(* IEC 61131-3 sources: F100R_S278_Temperville/MyController.device.xml.v3^/Plc Logic.plclogic.xml.v3^/Application.application.xml.v3^/02_Operação (part 3) *)

(* ---- K_Guilhotina01Inf.prg.st ---- *)
PROGRAM K_Guilhotina01Inf
VAR
	PassoHomeGuilhotina01Inf: INT;
	PassoAjusteGuilhotina01Inf: INT;
	PassoPausaHomeGuilhotina01Inf: INT;
	PassoPausaAjusteGuilhotina01Inf: INT;
	PassoAlmHomeGuilhotina01Inf: INT;
	PassoAlmAjusteGuilhotina01Inf: INT;
	///Bloco Converte Milimetro em Pulsos
	ConversorMilimPul01Guilho01Inf: MmConversorPulso;
	///Bloco Converte Milimetro em Pulsos
	ConversorMilimPul02Guilho01Inf: MmConversorPulso;
	///Bloco Converte Pulsos em Milimetros
	ConversorPulMilimGuilho01Inf: PulsoConversorMm;
	xSetValorSpAltGuil01InfSup: BOOL;
	iAlturaGhilhotina01InfAux: INT;
	xAjustarAlturaGuilhotina01Inf: BOOL;
	iVelocidadeHomeGuilhotina01Inf: INT;
	iVelocidadeGuilhotina01Inf: INT;
	dValEncoAlturaGuilhotina01Inf: DINT;
	dValEncoToleranciaGuilhotina01Inf: DINT;
	dValEncoAlturaVelMinGuilhotina01Inf: DINT;
	xAbreJogGuilhotina01Inf: BOOL;
	xFechaJogGuilhotina01Inf: BOOL;
	xAbreGuilhotina01Inf: BOOL;
	xFechaGuilhotina01Inf: BOOL;
END_VAR

IF iAlturaGhilhotina01Inf <> iAlturaGhilhotina01InfAux THEN
	xSetValorSpAltGuil01InfSup:=TRUE;

END_IF;

IF xSetValorSpAltGuil01InfSup THEN
	iAlturaGhilhotina01InfAux:=iAlturaGhilhotina01Inf;
ELSE
	IF NOT xMotorGuilhotina01InfLigado THEN
		iAlturaGhilhotina01Inf:=iAlturaAtualGuilhotina01Inf;
	END_IF;
END_IF

IF iAlturaGhilhotina01InfAux=iAlturaAtualGuilhotina01Inf THEN
	xSetValorSpAltGuil01InfSup:=FALSE;
END_IF

// CONVERSÃO MILIMETROS EM PULSOS

ConversorMilimPul01Guilho01Inf(
	dPulso:= 105563,
	dMilimetro:= 100,
	iEntrMilimetro01:= iAlturaGhilhotina01InfAux,//iAlturaGhilhotina02,
	dSaidaPulso01=> dValEncoAlturaGuilhotina01Inf);

ConversorMilimPul02Guilho01Inf(
	dPulso:= 105563,
	dMilimetro:= 100,
	iEntrMilimetro01:= 2,//iValEncoToleranciaGuilhotina,
	iEntrMilimetro02:= 8,//iValEncoAlturaVelMinGuilhotina,
	dSaidaPulso01=> dValEncoToleranciaGuilhotina01Inf,
	dSaidaPulso02=> dValEncoAlturaVelMinGuilhotina01Inf);

// SEQUENCIA DE HOME

CASE PassoHomeGuilhotina01Inf OF

		0:	IF xIniciaHomeGuilhotina01Inf THEN
				PassoHomeGuilhotina01Inf:=10;
			END_IF

		10:	xIniciaHomeGuilhotina01Inf:=FALSE;
			xHomeGuilhotina01InfOk:=FALSE;
			xAjusteAlturaGuilhotina01InfOK:=FALSE;
			xGuilhotina01InfEmHome:=TRUE;
			iVelocidadeGuilhotina01Inf:= 300;//1*iVelocidadeHomeDuctosResfrSup02;
			PassoHomeGuilhotina01Inf:=15;

		15: xFechaGuilhotina01Inf:=TRUE;
			PassoHomeGuilhotina01Inf:=20;

		20:	IF xSensorFechadoGuilhotina01Inf THEN
				PassoHomeGuilhotina01Inf:=50;
			END_IF
			IF xPause THEN
				PassoPausaHomeGuilhotina01Inf:=10;
				PassoHomeGuilhotina01Inf:=300;
			END_IF
			IF xAlarmeMotorGuilhotina01Inf THEN
				PassoAlmHomeGuilhotina01Inf:=10;
				PassoHomeGuilhotina01Inf:=400;
			END_IF

		50:	xFechaGuilhotina01Inf:=FALSE;
			PassoHomeGuilhotina01Inf:=55;

		55:	iVelocidadeGuilhotina01Inf:= 50;
			PassoHomeGuilhotina01Inf:=56;

		56:	xAbreGuilhotina01Inf:=TRUE;
			PassoHomeGuilhotina01Inf:=60;

		60:	IF NOT xSensorFechadoGuilhotina01Inf THEN
				PassoHomeGuilhotina01Inf:=70;
			END_IF
			IF xPause THEN
				PassoPausaHomeGuilhotina01Inf:=50;
				PassoHomeGuilhotina01Inf:=300;
			END_IF
			IF xAlarmeMotorGuilhotina01Inf THEN
				PassoAlmHomeGuilhotina01Inf:=50;
				PassoHomeGuilhotina01Inf:=400;
			END_IF

		70:	xAbreGuilhotina01Inf:=FALSE;
			PassoHomeGuilhotina01Inf:=74;

		74:	IF NOT xMotorGuilhotina01InfLigado THEN
				PassoHomeGuilhotina01Inf:=75;
			END_IF

		75: xHomeEncoderGuilhotinaResfriador01Inf:=TRUE;
			PassoHomeGuilhotina01Inf:=80;

		80: xHomeEncoderGuilhotinaResfriador01Inf:=FALSE;
			xGuilhotina01InfEmHome:=FALSE;
			xHomeGuilhotina01InfOk:=TRUE;

		// Emergência Pausa/Reinicio
		300:xAbreGuilhotina01Inf:=FALSE;
			xAbreGuilhotina01Inf:=FALSE;
			PassoHomeGuilhotina01Inf:=301;

		301:xDuctosSup02EmHome:=FALSE;
			PassoHomeGuilhotina01Inf:=302;

		302:IF xRestart THEN
				PassoHomeGuilhotina01Inf:=303;
			END_IF

		303:PassoHomeGuilhotina01Inf:=0;//PassoPausaHomeDuctosResfrSup02;

		// Alarme Motor Parada/Reinicio
		400:xFechaGuilhotina01Inf:=FALSE;
			xAbreGuilhotina01Inf:=FALSE;
			PassoHomeGuilhotina01Inf:=401;

		401:PassoHomeGuilhotina01Inf:=402;

		402:IF xRestart AND iCanOpenInverGuilResfr01InfStateOk THEN
				PassoHomeGuilhotina01Inf:=PassoAlmHomeGuilhotina01Inf;
			END_IF
END_CASE

// SEQUENCIA DE FUNCIONAMENTO

IF (xBtRecAjustaGuilhotina01Inf OR BtParamGuilhotina01Inf) AND xHomeGuilhotina01InfOk THEN
	xAjustarAlturaGuilhotina01Inf:=TRUE;
	xBtRecAjustaGuilhotina01Inf:=FALSE;
	BtParamGuilhotina01Inf:=FALSE;
ELSE
	xBtRecAjustaGuilhotina01Inf:=FALSE;
	BtParamGuilhotina01Inf:=FALSE;
END_IF

CASE PassoAjusteGuilhotina01Inf OF

		0:	IF xAjustarAlturaGuilhotina01Inf THEN
				PassoAjusteGuilhotina01Inf:=10;
			END_IF

		10:	xAjustarAlturaGuilhotina01Inf:=FALSE;
			xAjusteAlturaGuilhotina01InfOK:=FALSE;
			xGuilhotina01InfEmAjuste:=TRUE;
			IF (dValorEncoderGuilhotinaResfriador01Inf>=dValEncoAlturaGuilhotina01Inf-dValEncoToleranciaGuilhotina01Inf) AND (dValorEncoderGuilhotinaResfriador01Inf<=dValEncoAlturaGuilhotina01Inf+dValEncoToleranciaGuilhotina01Inf) THEN
				PassoAjusteGuilhotina01Inf:=180;//Não se Move
			END_IF
			IF dValorEncoderGuilhotinaResfriador01Inf<dValEncoAlturaGuilhotina01Inf-dValEncoToleranciaGuilhotina01Inf THEN
				PassoAjusteGuilhotina01Inf:=20;//Sobe
			END_IF
			IF dValorEncoderGuilhotinaResfriador01Inf>dValEncoAlturaGuilhotina01Inf+dValEncoToleranciaGuilhotina01Inf THEN
				PassoAjusteGuilhotina01Inf:=100;//Desce
			END_IF

//Sobe

		20:	iVelocidadeGuilhotina01Inf:= iVelocidadeAjusteGuilhotina01Inf;
			PassoAjusteGuilhotina01Inf:=25;

		25: xAbreGuilhotina01Inf:=TRUE;
			PassoAjusteGuilhotina01Inf:=30;

		30:	IF dValorEncoderGuilhotinaResfriador01Inf>=dValEncoAlturaGuilhotina01Inf-dValEncoAlturaVelMinGuilhotina01Inf THEN
				PassoAjusteGuilhotina01Inf:=40;
			END_IF
			IF iVelocidadeGuilhotina01Inf<> iVelocidadeAjusteGuilhotina01Inf THEN
				PassoAjusteGuilhotina01Inf:=20;
			END_IF
			IF xSensorAbertoGuilhotina01Inf THEN
				PassoAjusteGuilhotina01Inf:=200;
			END_IF

			IF xPause THEN
				PassoPausaAjusteGuilhotina01Inf:=20;
				PassoAjusteGuilhotina01Inf:=300;
			END_IF
			IF xAlarmeMotorGuilhotina01Inf THEN
				PassoAlmAjusteGuilhotina01Inf:=20;
				PassoAjusteGuilhotina01Inf:=400;
			END_IF

		40:	iVelocidadeGuilhotina01Inf:= iVelocidadeMinimaGuilhotina01Inf;
			PassoAjusteGuilhotina01Inf:=50;

		50:	IF dValorEncoderGuilhotinaResfriador01Inf>=dValEncoAlturaGuilhotina01Inf THEN
				PassoAjusteGuilhotina01Inf:=60;
			END_IF
			IF iVelocidadeGuilhotina01Inf<> iVelocidadeMinimaGuilhotina01Inf THEN
				PassoAjusteGuilhotina01Inf:=40;
			END_IF
			IF xPause THEN
				PassoPausaAjusteGuilhotina01Inf:=40;
				PassoAjusteGuilhotina01Inf:=300;
			END_IF
			IF xAlarmeMotorGuilhotina01Inf THEN
				PassoAlmAjusteGuilhotina01Inf:=40;
				PassoAjusteGuilhotina01Inf:=400;
			END_IF

		60: xAbreGuilhotina01Inf:=FALSE;
			PassoAjusteGuilhotina01Inf:=180;
//Desce

		100:iVelocidadeGuilhotina01Inf:= 1*iVelocidadeAjusteGuilhotina01Inf;
			PassoAjusteGuilhotina01Inf:=105;

		105:xFechaGuilhotina01Inf:=TRUE;
			PassoAjusteGuilhotina01Inf:=110;

		110:IF dValorEncoderGuilhotinaResfriador01Inf<dValEncoAlturaGuilhotina01Inf+dValEncoAlturaVelMinGuilhotina01Inf THEN
				PassoAjusteGuilhotina01Inf:=120;
			END_IF
			IF iVelocidadeGuilhotina01Inf<> 1*iVelocidadeAjusteGuilhotina01Inf THEN
				PassoAjusteGuilhotina01Inf:=100;
			END_IF
			IF	xSensorFechadoGuilhotina01Inf THEN
				PassoAjusteGuilhotina01Inf:=200;
			END_IF
			IF xPause THEN
				PassoPausaAjusteGuilhotina01Inf:=100;
				PassoAjusteGuilhotina01Inf:=300;
			END_IF
			IF xAlarmeMotorGuilhotina01Inf THEN
				PassoAlmAjusteGuilhotina01Inf:=100;
				PassoAjusteGuilhotina01Inf:=400;
			END_IF

		120:iVelocidadeGuilhotina01Inf:= 1*iVelocidadeMinimaGuilhotina01Inf;
			PassoAjusteGuilhotina01Inf:=130;

		130:IF  dValorEncoderGuilhotinaResfriador01Inf<=dValEncoAlturaGuilhotina01Inf THEN
				PassoAjusteGuilhotina01Inf:=140;
			END_IF
			IF xPause THEN
				PassoPausaAjusteGuilhotina01Inf:=120;
				PassoAjusteGuilhotina01Inf:=300;
			END_IF
			IF xAlarmeMotorGuilhotina01Inf THEN
				PassoAlmAjusteGuilhotina01Inf:=120;
				PassoAjusteGuilhotina01Inf:=400;
			END_IF

		140:xFechaGuilhotina01Inf:=FALSE;
			PassoAjusteGuilhotina01Inf:=180;
//Fim

		180:xAjusteAlturaGuilhotina01InfOK:=TRUE;
			xGuilhotina01InfEmAjuste:=FALSE;
			PassoAjusteGuilhotina01Inf:=0;

		200:xAbreGuilhotina01Inf:=FALSE;
			xFechaGuilhotina01Inf:=FALSE;
			PassoAjusteGuilhotina01Inf:=0;

		// Emergência Pausa/Reinicio
		300:xAbreGuilhotina01Inf:=FALSE;
			xFechaGuilhotina01Inf:=FALSE;
			PassoAjusteGuilhotina01Inf:=301;

		301:PassoAjusteGuilhotina01Inf:=302;

		302:IF xRestart THEN
				PassoAjusteGuilhotina01Inf:=303;
			END_IF

		303: PassoAjusteGuilhotina01Inf:=PassoPausaAjusteGuilhotina01Inf;

		// Alarme Motor Parada/Reinicio
		400:xAbreGuilhotina01Inf:=FALSE;
			xFechaGuilhotina01Inf:=FALSE;
			PassoAjusteGuilhotina01Inf:=401;

		401:PassoAjusteGuilhotina01Inf:=402;

		402:IF xRestart AND iCanOpenInverGuilResfr01InfStateOk THEN
				PassoAjusteGuilhotina01Inf:=PassoAlmAjusteGuilhotina01Inf;
			END_IF

END_CASE

// MOVIMENTAÇÃO PELO COMANDO ENTRADAS DIGITAIS DO INVERSOR
// Comando e Dirreção
xMotorGuilhotina01InfAbre:= xAbreGuilhotina01Inf OR xAbreJogGuilhotina01Inf;
xMotorGuilhotina01InfFecha:= xFechaGuilhotina01Inf OR xFechaJogGuilhotina01Inf;

InversorGuilhot01Inf.i_xAvanco:=xMotorGuilhotina01InfAbre;
InversorGuilhot01Inf.i_xRecuo:=xMotorGuilhotina01InfFecha;

// Velocidade
InversorGuilhot01Inf.i_iFreqRef:=iVelocidadeGuilhotina01Inf;
//---------------------------------------------------------------------------------\\

ConversorPulMilimGuilho01Inf(
	dPulso:=105563,
	dMilimetro:= 100,
	dEntradaPulso01:= dValorEncoderGuilhotinaResfriador01Inf,
	iSaidaMilimetro01=> iAlturaAtualGuilhotina01Inf );

IF xOperacaoManual THEN
	PassoHomeGuilhotina01Inf:=0;
	PassoAjusteGuilhotina01Inf:=0;
	xIniciaHomeGuilhotina01Inf:=FALSE;
	xAjusteAlturaGuilhotina01InfOK:=FALSE;
	xGuilhotina01InfEmHome:=FALSE;
	xGuilhotina01InfEmAjuste:=FALSE;

	xAbreGuilhotina01Inf:=FALSE;
	xFechaGuilhotina01Inf:=FALSE;
END_IF

(*-------------------- Manual Jog--------------------------*)

(* ---- K_Guilhotina01Sup.prg.st ---- *)
PROGRAM K_Guilhotina01Sup
VAR
	PassoHomeGuilhotina01Sup: INT;
	PassoAjusteGuilhotina01Sup: INT;
	PassoPausaHomeGuilhotina01Sup: INT;
	PassoPausaAjusteGuilhotina01Sup: INT;
	PassoAlmHomeGuilhotina01Sup: INT;
	PassoAlmAjusteGuilhotina01Sup: INT;
	///Bloco Converte Milimetro em Pulsos
	ConversorMilimPul01Guilho01Sup: MmConversorPulso;
	///Bloco Converte Milimetro em Pulsos
	ConversorMilimPul02Guilho01Sup: MmConversorPulso;
	///Bloco Converte Pulsos em Milimetros
	ConversorPulMilimGuilho01Sup: PulsoConversorMm;
	xSetValorSpAltGuil01SupSup: BOOL;
	iAlturaGhilhotina01SupAux: INT;
	xAjustarAlturaGuilhotina01Sup: BOOL;
	iVelocidadeHomeGuilhotina01Sup: INT;
	iVelocidadeGuilhotina01Sup: INT;
	dValEncoAlturaGuilhotina01Sup: DINT;
	dValEncoToleranciaGuilhotina01Sup: DINT;
	dValEncoAlturaVelMinGuilhotina01Sup: DINT;
	xAbreJogGuilhotina01Sup: BOOL;
	xFechaJogGuilhotina01Sup: BOOL;
	xAbreGuilhotina01Sup: BOOL;
	xFechaGuilhotina01Sup: BOOL;
END_VAR

IF iAlturaGhilhotina01Sup <> iAlturaGhilhotina01SupAux THEN
	xSetValorSpAltGuil01SupSup:=TRUE;

END_IF;

IF xSetValorSpAltGuil01SupSup THEN
	iAlturaGhilhotina01SupAux:=iAlturaGhilhotina01Sup;
ELSE
	IF NOT xMotorGuilhotina01SupLigado THEN
		iAlturaGhilhotina01Sup:=iAlturaAtualGuilhotina01Sup;
	END_IF;
END_IF

IF iAlturaGhilhotina01SupAux=iAlturaAtualGuilhotina01Sup THEN
	xSetValorSpAltGuil01SupSup:=FALSE;
END_IF

// CONVERSÃO MILIMETROS EM PULSOS

ConversorMilimPul01Guilho01Sup(
	dPulso:= 107918,
	dMilimetro:= 100,
	iEntrMilimetro01:= iAlturaGhilhotina01SupAux,//iAlturaGhilhotina02,
	dSaidaPulso01=> dValEncoAlturaGuilhotina01Sup);

ConversorMilimPul02Guilho01Sup(
	dPulso:= 107918,
	dMilimetro:= 100,
	iEntrMilimetro01:= 2,//iValEncoToleranciaGuilhotina,
	iEntrMilimetro02:= 8,//iValEncoAlturaVelMinGuilhotina,
	dSaidaPulso01=> dValEncoToleranciaGuilhotina01Sup,
	dSaidaPulso02=> dValEncoAlturaVelMinGuilhotina01Sup);

// SEQUENCIA DE HOME

CASE PassoHomeGuilhotina01Sup OF

		0:	IF xIniciaHomeGuilhotina01Sup THEN
				PassoHomeGuilhotina01Sup:=10;
			END_IF

		10:	xIniciaHomeGuilhotina01Sup:=FALSE;
			xHomeGuilhotina01SupOk:=FALSE;
			xAjusteAlturaGuilhotina01SupOK:=FALSE;
			xGuilhotina01SupEmHome:=TRUE;
			iVelocidadeGuilhotina01Sup:= 300;//1*iVelocidadeHomeDuctosResfrSup02;
			PassoHomeGuilhotina01Sup:=15;

		15: xFechaGuilhotina01Sup:=TRUE;
			PassoHomeGuilhotina01Sup:=20;

		20:	IF xSensorFechadoGuilhotina01Sup THEN
				PassoHomeGuilhotina01Sup:=50;
			END_IF
			IF xPause THEN
				PassoPausaHomeGuilhotina01Sup:=10;
				PassoHomeGuilhotina01Sup:=300;
			END_IF
			IF xAlarmeMotorGuilhotina01Sup THEN
				PassoAlmHomeGuilhotina01Sup:=10;
				PassoHomeGuilhotina01Sup:=400;
			END_IF

		50:	xFechaGuilhotina01Sup:=FALSE;
			PassoHomeGuilhotina01Sup:=55;

		55:	iVelocidadeGuilhotina01Sup:= 50;
			PassoHomeGuilhotina01Sup:=56;

		56:	xAbreGuilhotina01Sup:=TRUE;
			PassoHomeGuilhotina01Sup:=60;

		60:	IF NOT xSensorFechadoGuilhotina01Sup THEN
				PassoHomeGuilhotina01Sup:=70;
			END_IF
			IF xPause THEN
				PassoPausaHomeGuilhotina01Sup:=50;
				PassoHomeGuilhotina01Sup:=300;
			END_IF
			IF xAlarmeMotorGuilhotina01Sup THEN
				PassoAlmHomeGuilhotina01Sup:=50;
				PassoHomeGuilhotina01Sup:=400;
			END_IF

		70:	xAbreGuilhotina01Sup:=FALSE;
			PassoHomeGuilhotina01Sup:=74;

		74:	IF NOT xMotorGuilhotina01SupLigado THEN
				PassoHomeGuilhotina01Sup:=75;
			END_IF

		75: xHomeEncoderGuilhotinaResfriador01Sup:=TRUE;
			PassoHomeGuilhotina01Sup:=80;

		80: xHomeEncoderGuilhotinaResfriador01Sup:=FALSE;
			xGuilhotina01SupEmHome:=FALSE;
			xHomeGuilhotina01SupOk:=TRUE;

		// Emergência Pausa/Reinicio
		300:xAbreGuilhotina01Sup:=FALSE;
			xAbreGuilhotina01Sup:=FALSE;
			PassoHomeGuilhotina01Sup:=301;

		301:xDuctosSup02EmHome:=FALSE;
			PassoHomeGuilhotina01Sup:=302;

		302:IF xRestart THEN
				PassoHomeGuilhotina01Sup:=303;
			END_IF

		303:PassoHomeGuilhotina01Sup:=0;//PassoPausaHomeDuctosResfrSup02;

		// Alarme Motor Parada/Reinicio
		400:xFechaGuilhotina01Sup:=FALSE;
			xAbreGuilhotina01Sup:=FALSE;
			PassoHomeGuilhotina01Sup:=401;

		401:PassoHomeGuilhotina01Sup:=402;

		402:IF xRestart AND iCanOpenInverGuilResfr01SupStateOk THEN
				PassoHomeGuilhotina01Sup:=PassoAlmHomeGuilhotina01Sup;
			END_IF
END_CASE

// SEQUENCIA DE FUNCIONAMENTO

IF (xBtRecAjustaGuilhotina01Sup OR BtParamGuilhotina01Sup) AND xHomeGuilhotina01SupOk THEN
	xAjustarAlturaGuilhotina01Sup:=TRUE;
	xBtRecAjustaGuilhotina01Sup:=FALSE;
	BtParamGuilhotina01Sup:=FALSE;
ELSE
	xBtRecAjustaGuilhotina01Sup:=FALSE;
	BtParamGuilhotina01Sup:=FALSE;
END_IF

CASE PassoAjusteGuilhotina01Sup OF

		0:	IF xAjustarAlturaGuilhotina01Sup THEN
				PassoAjusteGuilhotina01Sup:=10;
			END_IF

		10:	xAjustarAlturaGuilhotina01Sup:=FALSE;
			xAjusteAlturaGuilhotina01SupOK:=FALSE;
			xGuilhotina01SupEmAjuste:=TRUE;
			IF (dValorEncoderGuilhotinaResfriador01Sup>=dValEncoAlturaGuilhotina01Sup-dValEncoToleranciaGuilhotina01Sup) AND (dValorEncoderGuilhotinaResfriador01Sup<=dValEncoAlturaGuilhotina01Sup+dValEncoToleranciaGuilhotina01Sup) THEN
				PassoAjusteGuilhotina01Sup:=180;//Não se Move
			END_IF
			IF dValorEncoderGuilhotinaResfriador01Sup<dValEncoAlturaGuilhotina01Sup-dValEncoToleranciaGuilhotina01Sup THEN
				PassoAjusteGuilhotina01Sup:=20;//Sobe
			END_IF
			IF dValorEncoderGuilhotinaResfriador01Sup>dValEncoAlturaGuilhotina01Sup+dValEncoToleranciaGuilhotina01Sup THEN
				PassoAjusteGuilhotina01Sup:=100;//Desce
			END_IF

//Sobe

		20:	iVelocidadeGuilhotina01Sup:= iVelocidadeAjusteGuilhotina01Sup;
			PassoAjusteGuilhotina01Sup:=25;

		25: xAbreGuilhotina01Sup:=TRUE;
			PassoAjusteGuilhotina01Sup:=30;

		30:	IF dValorEncoderGuilhotinaResfriador01Sup>=dValEncoAlturaGuilhotina01Sup-dValEncoAlturaVelMinGuilhotina01Sup THEN
				PassoAjusteGuilhotina01Sup:=40;
			END_IF
			IF iVelocidadeGuilhotina01Sup<> iVelocidadeAjusteGuilhotina01Sup THEN
				PassoAjusteGuilhotina01Sup:=20;
			END_IF
			IF xSensorAbertoGuilhotina01Sup THEN
				PassoAjusteGuilhotina01Sup:=200;
			END_IF

			IF xPause THEN
				PassoPausaAjusteGuilhotina01Sup:=20;
				PassoAjusteGuilhotina01Sup:=300;
			END_IF
			IF xAlarmeMotorGuilhotina01Sup THEN
				PassoAlmAjusteGuilhotina01Sup:=20;
				PassoAjusteGuilhotina01Sup:=400;
			END_IF

		40:	iVelocidadeGuilhotina01Sup:= iVelocidadeMinimaGuilhotina01Sup;
			PassoAjusteGuilhotina01Sup:=50;

		50:	IF dValorEncoderGuilhotinaResfriador01Sup>=dValEncoAlturaGuilhotina01Sup THEN
				PassoAjusteGuilhotina01Sup:=60;
			END_IF
			IF iVelocidadeGuilhotina01Sup<> iVelocidadeMinimaGuilhotina01Sup THEN
				PassoAjusteGuilhotina01Sup:=40;
			END_IF
			IF xPause THEN
				PassoPausaAjusteGuilhotina01Sup:=40;
				PassoAjusteGuilhotina01Sup:=300;
			END_IF
			IF xAlarmeMotorGuilhotina01Sup THEN
				PassoAlmAjusteGuilhotina01Sup:=40;
				PassoAjusteGuilhotina01Sup:=400;
			END_IF

		60: xAbreGuilhotina01Sup:=FALSE;
			PassoAjusteGuilhotina01Sup:=180;
//Desce

		100:iVelocidadeGuilhotina01Sup:= 1*iVelocidadeAjusteGuilhotina01Sup;
			PassoAjusteGuilhotina01Sup:=105;

		105:xFechaGuilhotina01Sup:=TRUE;
			PassoAjusteGuilhotina01Sup:=110;

		110:IF dValorEncoderGuilhotinaResfriador01Sup<dValEncoAlturaGuilhotina01Sup+dValEncoAlturaVelMinGuilhotina01Sup THEN
				PassoAjusteGuilhotina01Sup:=120;
			END_IF
			IF iVelocidadeGuilhotina01Sup<> 1*iVelocidadeAjusteGuilhotina01Sup THEN
				PassoAjusteGuilhotina01Sup:=100;
			END_IF
			IF	xSensorFechadoGuilhotina01Sup THEN
				PassoAjusteGuilhotina01Sup:=200;
			END_IF
			IF xPause THEN
				PassoPausaAjusteGuilhotina01Sup:=100;
				PassoAjusteGuilhotina01Sup:=300;
			END_IF
			IF xAlarmeMotorGuilhotina01Sup THEN
				PassoAlmAjusteGuilhotina01Sup:=100;
				PassoAjusteGuilhotina01Sup:=400;
			END_IF

		120:iVelocidadeGuilhotina01Sup:= 1*iVelocidadeMinimaGuilhotina01Sup;
			PassoAjusteGuilhotina01Sup:=130;

		130:IF  dValorEncoderGuilhotinaResfriador01Sup<=dValEncoAlturaGuilhotina01Sup THEN
				PassoAjusteGuilhotina01Sup:=140;
			END_IF
			IF xPause THEN
				PassoPausaAjusteGuilhotina01Sup:=120;
				PassoAjusteGuilhotina01Sup:=300;
			END_IF
			IF xAlarmeMotorGuilhotina01Sup THEN
				PassoAlmAjusteGuilhotina01Sup:=120;
				PassoAjusteGuilhotina01Sup:=400;
			END_IF

		140:xFechaGuilhotina01Sup:=FALSE;
			PassoAjusteGuilhotina01Sup:=180;
//Fim

		180:xAjusteAlturaGuilhotina01SupOK:=TRUE;
			xGuilhotina01SupEmAjuste:=FALSE;
			PassoAjusteGuilhotina01Sup:=0;

		200:xAbreGuilhotina01Sup:=FALSE;
			xFechaGuilhotina01Sup:=FALSE;
			PassoAjusteGuilhotina01Sup:=0;

		// Emergência Pausa/Reinicio
		300:xAbreGuilhotina01Sup:=FALSE;
			xFechaGuilhotina01Sup:=FALSE;
			PassoAjusteGuilhotina01Sup:=301;

		301:PassoAjusteGuilhotina01Sup:=302;

		302:IF xRestart THEN
				PassoAjusteGuilhotina01Sup:=303;
			END_IF

		303: PassoAjusteGuilhotina01Sup:=PassoPausaAjusteGuilhotina01Sup;

		// Alarme Motor Parada/Reinicio
		400:xAbreGuilhotina01Sup:=FALSE;
			xFechaGuilhotina01Sup:=FALSE;
			PassoAjusteGuilhotina01Sup:=401;

		401:PassoAjusteGuilhotina01Sup:=402;

		402:IF xRestart AND iCanOpenInverGuilResfr01SupStateOk THEN
				PassoAjusteGuilhotina01Sup:=PassoAlmAjusteGuilhotina01Sup;
			END_IF

END_CASE

// MOVIMENTAÇÃO PELO COMANDO ENTRADAS DIGITAIS DO INVERSOR
// Comando e Dirreção
xMotorGuilhotina01SupAbre:= xAbreGuilhotina01Sup OR xAbreJogGuilhotina01Sup;
xMotorGuilhotina01SupFecha:= xFechaGuilhotina01Sup OR xFechaJogGuilhotina01Sup;

InversorGuilhot01Sup.i_xAvanco:=xMotorGuilhotina01SupAbre;
InversorGuilhot01Sup.i_xRecuo:=xMotorGuilhotina01SupFecha;

// Velocidade
InversorGuilhot01Sup.i_iFreqRef:=iVelocidadeGuilhotina01Sup;
//---------------------------------------------------------------------------------\\

ConversorPulMilimGuilho01Sup(
	dPulso:=107918,
	dMilimetro:= 100,
	dEntradaPulso01:= dValorEncoderGuilhotinaResfriador01Sup,
	iSaidaMilimetro01=> iAlturaAtualGuilhotina01Sup );

IF xOperacaoManual THEN
	PassoHomeGuilhotina01Sup:=0;
	PassoAjusteGuilhotina01Sup:=0;
	xIniciaHomeGuilhotina01Sup:=FALSE;
	xAjusteAlturaGuilhotina01SupOK:=FALSE;
	xGuilhotina01SupEmHome:=FALSE;
	xGuilhotina01SupEmAjuste:=FALSE;

	xAbreGuilhotina01Sup:=FALSE;
	xFechaGuilhotina01Sup:=FALSE;
END_IF

(*-------------------- Manual Jog--------------------------*)

(* ---- K_Guilhotina02.prg.st ---- *)
PROGRAM K_Guilhotina02
VAR
	PassoHomeGuilhotina02: INT;
	PassoAjusteGuilhotina02: INT;
	PassoPausaHomeGuilhotina02: INT;
	PassoPausaAjusteGuilhotina02: INT;
	PassoAlmHomeGuilhotina02: INT;
	PassoAlmAjusteGuilhotina02: INT;
	xSinalAjusteG02: INT;
	ContadorEncoderPo: ContadorUpDown;
	TonHomeGuilho02: TON;
	xTonHomeGuilho02In: BOOL;
	xTonHomeGuilho02Q: BOOL;
	///Bloco Converte Milimetro em Pulsos
	ConversorMilimPul01Guilho02: MmConversorPulso;
	///Bloco Converte Milimetro em Pulsos
	ConversorMilimPul02Guilho02: MmConversorPulso;
	///Bloco Converte Pulsos em Milimetros
	ConversorPulMilimGuilho02: PulsoConversorMm;
	xExecutaMovGuilhotina02: BOOL;
	xExecutaStopGuilhotina02: BOOL;
	xStopGuilhotina02Done: BOOL;
	xSetValorSpAltGuil02Sup: BOOL;
	iAlturaGhilhotina02Aux: INT;
	xAjustarAlturaGuilhotina02: BOOL;
	iVelocidadeHomeGuilhotina02: INT;
	iVelocidadeGuilhotina02: INT;
	dValEncoAlturaGuilhotina02: DINT;
	dValEncoToleranciaGuilhotina02: DINT;
	dValEncoAlturaVelMinGuilhotina02: DINT;
	xCmdPositivoGuilhotina02: BOOL;
	xCmdNegativoGuilhotina02: BOOL;
	xIncrementaEncoderGuilhotina02Po: BOOL;
	xDecrementaEncoderGuilhotina02Po: BOOL;
	iValorEncoderGuilhotina02Po: INT;
	xSobeJogGuilhotina02: BOOL;
	xDesceJogGuilhotina02: BOOL;
	xSobeGuilhotina02: BOOL;
	xDesceGuilhotina02: BOOL;

END_VAR

IF iAlturaGhilhotina02 <> iAlturaGhilhotina02Aux THEN
	xSetValorSpAltGuil02Sup:=TRUE;

END_IF;

IF xSetValorSpAltGuil02Sup THEN
	iAlturaGhilhotina02Aux:=iAlturaGhilhotina02;
ELSE
	IF NOT xMotorGuilhotina02Ligado THEN
		iAlturaGhilhotina02:=iAlturaAtualGuilhotina02;
	END_IF;
END_IF

IF iAlturaGhilhotina02Aux=iAlturaAtualGuilhotina02 THEN
	xSetValorSpAltGuil02Sup:=FALSE;
END_IF

// CONVERSÃO MILIMETROS EM PULSOS

ConversorMilimPul01Guilho02(
	dPulso:= 234600,
	dMilimetro:= 100,
	iEntrMilimetro01:= iAlturaGhilhotina02Aux,//iAlturaGhilhotina02,
	dSaidaPulso01=> dValEncoAlturaGuilhotina02);

ConversorMilimPul02Guilho02(
	dPulso:= 234600,
	dMilimetro:= 100,
	iEntrMilimetro01:= 2,//iValEncoToleranciaGuilhotina,
	iEntrMilimetro02:= 4,//iValEncoAlturaVelMinGuilhotina,
	dSaidaPulso01=> dValEncoToleranciaGuilhotina02,
	dSaidaPulso02=> dValEncoAlturaVelMinGuilhotina02);

// SEQUENCIA DE HOME

CASE PassoHomeGuilhotina02 OF

		0:	IF xIniciaHomeGuilhotina02(* OR xAutoHomeGuilho02*) THEN
				PassoHomeGuilhotina02:=5;
			END_IF

		5:	xIniciaHomeGuilhotina02:=FALSE;
			xAutoHomeGuilho02:=FALSE;
			xGuilhotina02EmAjuste:=FALSE;
			xHomeGuilhotina02Ok:=FALSE;
			xAjusteAlturaGuilhotina02OK:=FALSE;
			xGuilhotina02EmHome:=TRUE;
			PassoHomeGuilhotina02:=8;

		8: IF xSensorZeroGuilhotina02 THEN
				PassoHomeGuilhotina02:=9;
			ELSE
				PassoHomeGuilhotina02:=13;
			END_IF

		9: iVelocidadeGuilhotina02:= 600;//iVelocidadeHomeGuilhotina02;
		   PassoHomeGuilhotina02:=10;

		10:	xSobeGuilhotina02:=TRUE;
			PassoHomeGuilhotina02:=11;

		11: IF NOT xSensorZeroGuilhotina02 THEN
				PassoHomeGuilhotina02:=30;
			END_IF
			IF xPause THEN
				PassoPausaHomeGuilhotina02:=50;
				PassoHomeGuilhotina02:=300;
			END_IF
			IF xAlarmeMotorGuilhotina02 THEN
				PassoAlmHomeGuilhotina02:=50;
				PassoHomeGuilhotina02:=400;
			END_IF

		13:	PassoHomeGuilhotina02:=14;

		14:	iVelocidadeGuilhotina02:= 600;//iVelocidadeHomeGuilhotina02;
			xSinalAjusteG02:=1;
			PassoHomeGuilhotina02:=15;

		15:	xSobeGuilhotina02:=TRUE;
			PassoHomeGuilhotina02:=20;

		20:	IF xSensorPositivoGuilhotina02 THEN
				PassoHomeGuilhotina02:=30;
			END_IF
			IF xSensorZeroGuilhotina02 THEN
				PassoHomeGuilhotina02:=9;//50;
			END_IF
			IF xPause THEN
				PassoPausaHomeGuilhotina02:=15;
				PassoHomeGuilhotina02:=300;
			END_IF
			IF xAlarmeMotorGuilhotina02 THEN
				PassoAlmHomeGuilhotina02:=15;
				PassoHomeGuilhotina02:=400;
			END_IF

		30: xSobeGuilhotina02:=TRUE;
			PassoHomeGuilhotina02:=31;

		31:	iVelocidadeGuilhotina02:=-1*600;//iVelocidadeHomeGuilhotina02;
			xSinalAjusteG02:=-1;
			PassoHomeGuilhotina02:=40;

		40:	IF xSensorNegativoGuilhotina02 THEN
				PassoHomeGuilhotina02:=13;
			END_IF
			IF xSensorZeroGuilhotina02 THEN
				PassoHomeGuilhotina02:=50;
			END_IF
			IF xPause THEN
				PassoPausaHomeGuilhotina02:=30;
				PassoHomeGuilhotina02:=300;
			END_IF
			IF xAlarmeMotorGuilhotina02 THEN
				PassoAlmHomeGuilhotina02:=30;
				PassoHomeGuilhotina02:=400;
			END_IF

		50: iVelocidadeGuilhotina02:= xSinalAjusteG02*150;
			PassoHomeGuilhotina02:=53;

		53:	xTonHomeGuilho02In:=TRUE;
			PassoHomeGuilhotina02:=54;

		54: IF xTonHomeGuilho02Q THEN
				PassoHomeGuilhotina02:=60;
			END_IF

		60:	xTonHomeGuilho02In:=FALSE;
			PassoHomeGuilhotina02:=70;

		70: xSobeGuilhotina02:=FALSE;
			PassoHomeGuilhotina02:=80;

		80: xHomeEncoderGuilhotinaResfriador02:=TRUE;
			PassoHomeGuilhotina02:=81;

		81:PassoHomeGuilhotina02:=82;

		82: xHomeEncoderGuilhotinaResfriador02:=FALSE;
			PassoHomeGuilhotina02:=83;

		83:	xHomeGuilhotina02Ok:=TRUE;
			xGuilhotina02EmHome:=FALSE;
			PassoHomeGuilhotina02:=0;

		// Emergência Pausa/Reinicio
		300:xSobeGuilhotina02:=FALSE;
			xDesceGuilhotina02:=FALSE;
			PassoHomeGuilhotina02:=301;

		301:xGuilhotina02EmHome:=FALSE;
			PassoHomeGuilhotina02:=302;

		302:IF xRestart THEN
				PassoHomeGuilhotina02:=303;
			END_IF

		303:PassoHomeGuilhotina02:=0;//PassoPausaHomeGuilhotina;

		// Alarme Motor Parada/Reinicio
		400:xSobeGuilhotina02:=FALSE;
			xDesceGuilhotina02:=FALSE;
			PassoHomeGuilhotina02:=401;

		401:PassoHomeGuilhotina02:=402;

		402:IF xRestart AND iCanOpenInverGuilResfr02StateOk THEN
				PassoHomeGuilhotina02:=PassoAlmHomeGuilhotina02;
			END_IF

END_CASE

TonHomeGuilho02(IN:= xTonHomeGuilho02In, PT:=T#1720MS , Q=> xTonHomeGuilho02Q, ET=> );

// SEQUENCIA DE FUNCIONAMENTO

IF (xBtRecAjustaGuilhotina02 OR BtParamGuilhotina02) AND xHomeGuilhotina02Ok THEN
	xAjustarAlturaGuilhotina02:=TRUE;
	xBtRecAjustaGuilhotina02:=FALSE;
	BtParamGuilhotina02:=FALSE;
ELSE
	xBtRecAjustaGuilhotina02:=FALSE;
	BtParamGuilhotina02:=FALSE;
END_IF

CASE PassoAjusteGuilhotina02 OF

		0:	IF xAjustarAlturaGuilhotina02 THEN
				PassoAjusteGuilhotina02:=10;
			END_IF

		10:	xAjustarAlturaGuilhotina02:=FALSE;
			xAjusteAlturaGuilhotina02OK:=FALSE;
			xGuilhotina02EmAjuste:=TRUE;
			IF (dValorEncoderGuilhotinaResfriador02>=dValEncoAlturaGuilhotina02-dValEncoToleranciaGuilhotina02) AND (dValorEncoderGuilhotinaResfriador02<=dValEncoAlturaGuilhotina02+dValEncoToleranciaGuilhotina02) THEN
				PassoAjusteGuilhotina02:=180;//Não se Move
			END_IF
			IF dValorEncoderGuilhotinaResfriador02<dValEncoAlturaGuilhotina02-dValEncoToleranciaGuilhotina02 THEN
				PassoAjusteGuilhotina02:=20;//Sobe
			END_IF
			IF dValorEncoderGuilhotinaResfriador02>dValEncoAlturaGuilhotina02+dValEncoToleranciaGuilhotina02 THEN
				PassoAjusteGuilhotina02:=100;//Desce
			END_IF

//Sobe
		20:	iVelocidadeGuilhotina02:= iVelocidadeAjusteGuilhotina02;
			PassoAjusteGuilhotina02:=25;

		25: xSobeGuilhotina02:=TRUE;
			PassoAjusteGuilhotina02:=30;

		30:	IF dValorEncoderGuilhotinaResfriador02>=dValEncoAlturaGuilhotina02-dValEncoAlturaVelMinGuilhotina02 THEN
				PassoAjusteGuilhotina02:=40;
			END_IF
			IF iVelocidadeGuilhotina02<> iVelocidadeAjusteGuilhotina02 THEN
				PassoAjusteGuilhotina02:=20;
			END_IF
			IF xSensorPositivoGuilhotina02 THEN
				PassoAjusteGuilhotina02:=200;
			END_IF

			IF xPause THEN
				PassoPausaAjusteGuilhotina02:=20;
				PassoAjusteGuilhotina02:=300;
			END_IF
			IF xAlarmeMotorGuilhotina02 THEN
				PassoAlmAjusteGuilhotina02:=20;
				PassoAjusteGuilhotina02:=400;
			END_IF

		40:	iVelocidadeGuilhotina02:= iVelocidadeMinimaGuilhotina02;
			PassoAjusteGuilhotina02:=50;

		50:	IF dValorEncoderGuilhotinaResfriador02>=dValEncoAlturaGuilhotina02 THEN
				PassoAjusteGuilhotina02:=60;
			END_IF
			IF iVelocidadeGuilhotina02<> iVelocidadeMinimaGuilhotina02 THEN
				PassoAjusteGuilhotina02:=40;
			END_IF
			IF xPause THEN
				PassoPausaAjusteGuilhotina02:=40;
				PassoAjusteGuilhotina02:=300;
			END_IF
			IF xAlarmeMotorGuilhotina02 THEN
				PassoAlmAjusteGuilhotina02:=40;
				PassoAjusteGuilhotina02:=400;
			END_IF

		60: xSobeGuilhotina02:=FALSE;
			PassoAjusteGuilhotina02:=180;
//Desce

		100:iVelocidadeGuilhotina02:= 1*iVelocidadeAjusteGuilhotina02;
			PassoAjusteGuilhotina02:=105;

		105:xDesceGuilhotina02:=TRUE;
			PassoAjusteGuilhotina02:=110;

		110:IF dValorEncoderGuilhotinaResfriador02<dValEncoAlturaGuilhotina02+dValEncoAlturaVelMinGuilhotina02 THEN
				PassoAjusteGuilhotina02:=120;
			END_IF
			IF iVelocidadeGuilhotina02<> 1*iVelocidadeAjusteGuilhotina02 THEN
				PassoAjusteGuilhotina02:=100;
			END_IF
			IF	xSensorNegativoGuilhotina02 THEN
				PassoAjusteGuilhotina02:=200;
			END_IF
			IF xPause THEN
				PassoPausaAjusteGuilhotina02:=100;
				PassoAjusteGuilhotina02:=300;
			END_IF
			IF xAlarmeMotorGuilhotina02 THEN
				PassoAlmAjusteGuilhotina02:=100;
				PassoAjusteGuilhotina02:=400;
			END_IF

		120:iVelocidadeGuilhotina02:= 1*iVelocidadeMinimaGuilhotina02;
			PassoAjusteGuilhotina02:=130;

		130:IF  dValorEncoderGuilhotinaResfriador02<=dValEncoAlturaGuilhotina02 THEN
				PassoAjusteGuilhotina02:=140;
			END_IF
			IF xPause THEN
				PassoPausaAjusteGuilhotina02:=120;
				PassoAjusteGuilhotina02:=300;
			END_IF
			IF xAlarmeMotorGuilhotina02 THEN
				PassoAlmAjusteGuilhotina02:=120;
				PassoAjusteGuilhotina02:=400;
			END_IF

		140:xDesceGuilhotina02:=FALSE;
			PassoAjusteGuilhotina02:=180;
//Fim
		180:xExecutaStopGuilhotina02:=FALSE;
			xAjusteAlturaGuilhotina02OK:=TRUE;
			xGuilhotina02EmAjuste:=FALSE;
			PassoAjusteGuilhotina02:=0;

		200:xSobeGuilhotina02:=FALSE;
			xDesceGuilhotina02:=FALSE;
			PassoAjusteGuilhotina02:=0;

		// Emergência Pausa/Reinicio
		300:xSobeGuilhotina02:=FALSE;
			xDesceGuilhotina02:=FALSE;
			PassoAjusteGuilhotina02:=301;

		301:PassoAjusteGuilhotina02:=302;

		302:IF xRestart THEN
				PassoAjusteGuilhotina02:=303;
			END_IF

		303: PassoAjusteGuilhotina02:=PassoPausaAjusteGuilhotina02;

		// Alarme Motor Parada/Reinicio
		400:xSobeGuilhotina02:=FALSE;
			xDesceGuilhotina02:=FALSE;
			PassoAjusteGuilhotina02:=401;

		401:PassoAjusteGuilhotina02:=402;

		402:IF xRestart AND iCanOpenInverGuilResfr02StateOk THEN
				PassoAjusteGuilhotina02:=PassoAlmAjusteGuilhotina02;
			END_IF

END_CASE

// MOVIMENTAÇÃO PELO COMANDO ENTRADAS DIGITAIS DO INVERSOR
// Comando e Dirreção
xMotorGuilhotina02Sobe:= xSobeGuilhotina02 OR xSobeJogGuilhotina02;
xMotorGuilhotina02Desce:= xDesceGuilhotina02 OR xDesceJogGuilhotina02;

InversorGuilhot02.i_xAvanco:=xMotorGuilhotina02Sobe;
InversorGuilhot02.i_xRecuo:=xMotorGuilhotina02Desce;

// Velocidade
InversorGuilhot02.i_iFreqRef:=iVelocidadeGuilhotina02;
//---------------------------------------------------------------------------------\\

ConversorPulMilimGuilho02(
	dPulso:= 234600,
	dMilimetro:= 100,
	dEntradaPulso01:= dValorEncoderGuilhotinaResfriador02,
	iSaidaMilimetro01=> iAlturaAtualGuilhotina02 );

IF xOperacaoManual THEN
	PassoHomeGuilhotina02:=0;
	PassoAjusteGuilhotina02:=0;
	xIniciaHomeGuilhotina02:=FALSE;
	xAjusteAlturaGuilhotina02OK:=FALSE;
	xGuilhotina02EmHome:=FALSE;
	xGuilhotina02EmAjuste:=FALSE;

	xSobeGuilhotina02:=FALSE;
	xDesceGuilhotina02:=FALSE;
END_IF

(*-------------------- Manual Jog--------------------------*)

xSobeJogGuilhotina02:=xBtSobeGuilhtina02Manual AND NOT xSensorPositivoGuilhotina02 AND NOT xPausaEmergencia ;
xDesceJogGuilhotina02:=xBtDesceGuilhotina02Manual AND NOT xSensorNegativoGuilhotina02 AND NOT xPausaEmergencia ;

(* ---- L_EstagiosResfriador.prg.st ---- *)
PROGRAM L_EstagiosResfriador
VAR
	PassoEstagioResfriador: INT;
	///Bloco Conta Tempo de Pausa dos Roletes
	TimerTrocaEstagios1p2: Temporizador;
	///Bloco Conta Tempo de Pausa dos Roletes
	TimerTrocaEstagios2p3: Temporizador;
	///xIniciaTempoPrimeiroEstagio: BOOL;
	xFimTempoPrimeiroEstagio: BOOL;
	xFimTempoSegundoEstagio: BOOL;
END_VAR

// SEQUENCIA DE ESTAGIOS

CASE PassoEstagioResfriador OF

		0:	IF xInicioPrimeiroEstagio THEN //<- TASK/MesaResfriador
				PassoEstagioResfriador:=10;
			END_IF

		10:	xFimTrocaEstagiosResfriador:=FALSE;
			xInicioPrimeiroEstagio:=FALSE;
			xPrimeiroEstagioResfriador:=TRUE;
			//xIniciaTempoPrimeiroEstagio:=TRUE;
			PassoEstagioResfriador:=20;

		20:	IF xFimTempoPrimeiroEstagio OR xFimTrocaEstagiosResfriador THEN
				xInicioSegundoEstagio:=TRUE;
				PassoEstagioResfriador:=21;
			END_IF

		21: xInicioSegundoEstagio:=FALSE;
			PassoEstagioResfriador:=30;

		30:	xPrimeiroEstagioResfriador:=FALSE;
			xSegundoEstagioResfriador:=TRUE;
			//xLigaSegEstagDuctosSup01:= TRUE;
			//xLigaSegEstagDuctosInf01:= TRUE;
			xLigaSegEstagDuctosSup02:= TRUE;
			xLigaSegEstagDuctosInf02:= TRUE;
			//xSegundoEstagioVentilador01:=TRUE;
			//xSegundoEstagioVentilador02:=TRUE;
			xSegundoEstagioVentilador03:=TRUE;
			xSegundoEstagioVentilador04:=TRUE;
			PassoEstagioResfriador:=31;

		31:	IF xFimTempoSegundoEstagio OR xFimTrocaEstagiosResfriador THEN
				PassoEstagioResfriador:=32;
			END_IF

		32:	xSegundoEstagioResfriador:=FALSE;
			xTerceiroEstagioResfriador:=TRUE;
			//xLigaTerEstagDuctosSup01:= TRUE;
			//xLigaTerEstagDuctosInf01:= TRUE;
			xLigaTerEstagDuctosSup02:= TRUE;
			xLigaTerEstagDuctosInf02:= TRUE;
			//xTerceiroEstagioVentilador01:=TRUE;
			//xTerceiroEstagioVentilador02:=TRUE;
			xTerceiroEstagioVentilador03:=TRUE;
			xTerceiroEstagioVentilador04:=TRUE;
			PassoEstagioResfriador:=40;

		40:	IF xFimTrocaEstagiosResfriador THEN //<- TASK/MesaResfriador
				PassoEstagioResfriador:=50;
			END_IF

		50:	//xIniciaTempoPrimeiroEstagio:=FALSE;
			xTerceiroEstagioResfriador:=FALSE;
			xFimTempoPrimeiroEstagio:=FALSE;
			xFimTempoSegundoEstagio:=FALSE;
			xFimTrocaEstagiosResfriador:=FALSE;
			PassoEstagioResfriador:=0;

END_CASE

//TEMPORIZADOR TROCA DE ESTAGIOS DO RESFRIADOR
TimerTrocaEstagios1p2(
	IniciaTempo:= 	xInicioPrimeiroEstagio,
	AbortaTempo:= 	xOperacaoManual OR xFimTrocaEstagiosResfriador,
	SetPointTempo:= iTempoTrocaEstagioResfriamento,
	FimTempo:= 		xFimTempoPrimeiroEstagio,
	TempoDecorrido=>iTempoTrocaEstagioDecorrido ,
	TempoRestante=> );

TimerTrocaEstagios2p3(
	IniciaTempo:= 	xInicioSegundoEstagio,
	AbortaTempo:= 	xOperacaoManual OR xFimTrocaEstagiosResfriador,
	SetPointTempo:= iTempoTrocaEstagio02Resfriamento,
	FimTempo:= 		xFimTempoSegundoEstagio,
	TempoDecorrido=>iTempoTrocaEstagio02Decorrido ,
	TempoRestante=> );

IF xOperacaoManual THEN
	PassoEstagioResfriador:=0;
	xInicioPrimeiroEstagio:=FALSE;
	//xIniciaTempoPrimeiroEstagio:=FALSE;
	xPrimeiroEstagioResfriador:=FALSE;
	xSegundoEstagioResfriador:=FALSE;
	xTerceiroEstagioResfriador:=FALSE;
	xFimTempoPrimeiroEstagio:=FALSE;
	xFimTempoSegundoEstagio:=FALSE;
END_IF

(* ---- M_Ventilador01.prg.st ---- *)
PROGRAM M_Ventilador01
VAR
	PassoVentilador01: INT;
	PassoPauseVentilador01: INT;
	PassoAlmVentilador01: INT;
	PulsoLigaVentilador01: PulsoPositivo;
	iVelocidadeVentilador01: INT;
	xLigaVentilador01: BOOL;
	xFimVentilacao01: BOOL;
	xLigaTempoVentilador01: BOOL;
	xPulsoLigaVentilador01: BOOL;
	xLigaVent01SairForno: BOOL;
	xTempoMvVent01In: BOOL;
	xTempoMvVent01Q: BOOL;
	TempoMvVent01: ton;
	xLigaMotorVentilador01: BOOL;
	iVelocidadeVentilador01HZ: INT;
	dVelocidadeVentilador01HZ: DINT;
	rVelocidadeVentilador01HZ:REAL;
	rVelocidadeVentilador01 :REAL;
	PIDVENT01: FB_PID;

	rPidSaidaVent01	: REAL;
	iRefFreqVent01Pid	: INT ;

	xVentPassHabilitado	: BOOL ;
END_VAR

IF iVelocidade01Ventilador01<> 0 THEN
	xVentPassHabilitado:=TRUE;
ELSE
	xVentPassHabilitado:=FALSE;
END_IF

IF xEspessuraVidroFino THEN
	IF (iTempoAquecFornoRestante<=iTempoLigaVentilador01VidroFino) AND (iTempoAquecFornoRestante>0) AND xFornoEmCiclo AND xVentPassHabilitado THEN
		xLigaTempoVentilador01:=TRUE;
	ELSE
		xLigaTempoVentilador01:=FALSE;
	END_IF
ELSE
	IF (iTempoAquecFornoRestante<=iTempoLigaVentilador01VidroGros) AND (iTempoAquecFornoRestante>0) AND xFornoEmCiclo AND xVentPassHabilitado THEN
		xLigaTempoVentilador01:=TRUE;
	ELSE
		xLigaTempoVentilador01:=FALSE;
	END_IF
END_IF

xLigaVent01SairForno:=xSairForno AND xFornoEmCiclo and xFornoComCarga;

PulsoLigaVentilador01(Entrada:= xLigaTempoVentilador01 OR xLigaVent01SairForno OR xLigaVent01FimForno, SaidaPulsoPo=>xPulsoLigaVentilador01 );
IF xPulsoLigaVentilador01 THEN
	xLigaVentilador01:=TRUE;
	xFechaVenezVentPassV01:=TRUE;//-> TASK/T_VenezianaVentInfPass
END_IF

TempoMvVent01(IN:= xTempoMvVent01In, PT:=T#2S , Q=> xTempoMvVent01Q, ET=> );

// SEQUENCIA DE FUNCIONAMENTO
iVelocidade02Ventilador01:=iVelocidade01Ventilador01;
iVelocidade03Ventilador01:=iVelocidade01Ventilador01;

CASE PassoVentilador01 OF

		0:	IF xLigaVentilador01 THEN
				PassoVentilador01:=10;
			END_IF

		10:	xLigaVentilador01:=FALSE;
			xDesligaVentilador01:=FALSE;
			xDesligaFimVentilador01:=FALSE;
			xSegundoEstagioVentilador01:=FALSE;
			xTerceiroEstagioVentilador01:=FALSE;
			PassoVentilador01:=15;

		15:	xPrimeiroEstagioVentilador01:=TRUE;
			PassoVentilador01:=16;

		16:	IF  xSemEnergia THEN
				PassoVentilador01:=80;
			ELSIF xPause THEN
				PassoPauseVentilador01:=16;
				PassoVentilador01:=300;
			ELSIF xAlarmeMotorVentilador01 THEN
				PassoAlmVentilador01:=16;
				PassoVentilador01:=400;
			ELSE
				PassoVentilador01:=20;
			END_IF

		20:	iVelocidadeVentilador01:=iVelocidade01Ventilador01;
			PassoVentilador01:=21;

		21:	xLigaMotorVentilador01:=TRUE;
			PassoVentilador01:=22;

		22:	PassoVentilador01:=29;

		29:	PassoVentilador01:=59;//30; (* Alterado Ventilador tempera passagem*)

		// Fica Parado no passo 30 aguardando o inicio do segundo Estágio
		30:	IF iVelocidadeVentilador01<>iVelocidade01Ventilador01 THEN
				PassoVentilador01:=20;
			END_IF
			IF xSegundoEstagioVentilador01 THEN //<-TASK/EstagiosResfriador
				PassoVentilador01:=40;
			END_IF
			IF xDesligaVentilador01 THEN
				PassoVentilador01:=41;
			END_IF
			IF  xSemEnergia THEN
				PassoVentilador01:=80;
			END_IF
			IF xPause THEN
				PassoPauseVentilador01:=20;
				PassoVentilador01:=300;
			END_IF
			IF xAlarmeMotorVentilador01 THEN
				PassoAlmVentilador01:=20;
				PassoVentilador01:=400;
			END_IF

		40:	xSegundoEstagioVentilador01:=FALSE;
			xDesligaVentilador01:=FALSE; // Zera memoria desliga vent caso esteja em 1
			PassoVentilador01:=41;

		41:	xPrimeiroEstagioVentilador01:=FALSE;
			iVelocidadeVentilador01:=iVelocidade02Ventilador01;
			PassoVentilador01:=42;

		42:	PassoVentilador01:=43;

		43:	PassoVentilador01:=44;

		44:	PassoVentilador01:=50;
		// Fica Parado no Passo 50 aguardando o inicio do Terceiro Estágio
		50:	IF iVelocidadeVentilador01<>iVelocidade02Ventilador01 THEN
				PassoVentilador01:=41;
			END_IF
			IF xTerceiroEstagioVentilador01 THEN //<-TASK/EstagiosResfriador
				PassoVentilador01:=51;
			END_IF
			IF xDesligaVentilador01 THEN
				PassoVentilador01:=52;
			END_IF
			IF  xSemEnergia THEN
				PassoVentilador01:=80;
			END_IF
			IF xPause THEN
				PassoPauseVentilador01:=41;
				PassoVentilador01:=300;
			END_IF
			IF xAlarmeMotorVentilador01 THEN
				PassoAlmVentilador01:=41;
				PassoVentilador01:=400;
			END_IF

		51:	xTerceiroEstagioVentilador01:=FALSE;
			xDesligaVentilador01:=FALSE; // Zera memoria desliga vent caso esteja em 1
			PassoVentilador01:=52;

		52:	xSegundoEstagioVentilador01:=FALSE;
			iVelocidadeVentilador01:=iVelocidade03Ventilador01;
			PassoVentilador01:=53;

		53:	PassoVentilador01:=54;

		54:	PassoVentilador01:=55;

		55:	PassoVentilador01:=59;

			// Fica Parado no Passo 59 Aguardando
		59:	IF iVelocidadeVentilador01<>iVelocidade03Ventilador01 THEN
				PassoVentilador01:=20;//52; (* Alterador Tempera de passagem *)
			END_IF
			IF xLigaVentilador01 THEN
				PassoVentilador01:=10;
			END_IF
			IF xDesligaVentilador01 AND NOT xFornoEmEspera THEN
				PassoVentilador01:=60;
			END_IF
			IF xDesligaVentilador01 AND xFornoEmEspera THEN
				PassoVentilador01:=80;
			END_IF
			IF  xSemEnergia THEN
				PassoVentilador01:=80;
			END_IF
			IF xPause THEN
				PassoPauseVentilador01:=20;//52;
				PassoVentilador01:=300;
			END_IF
			IF xAlarmeMotorVentilador01 THEN
				PassoAlmVentilador01:=20;//52;
				PassoVentilador01:=400;
			END_IF

		60:	xDesligaVentilador01:=FALSE;
			xPrimeiroEstagioVentilador01:=FALSE;
			PassoVentilador01:=61;

		61:	IF iVelocidadeStbVentilador01<>0 THEN
				PassoVentilador01:=62;
			ELSE
				PassoVentilador01:=63;
			END_IF

		62:	xLigaMotorVentilador01:=TRUE;
			PassoVentilador01:=70;

		63:	xLigaMotorVentilador01:=FALSE;
			PassoVentilador01:=70;

		70:	iVelocidadeVentilador01:=iVelocidadeStbVentilador01;
			PassoVentilador01:=71;

		71:	IF iVelocidadeVentilador01<> iVelocidadeStbVentilador01 THEN
				PassoVentilador01:=61;
			END_IF
			IF xLigaVentilador01 THEN
				PassoVentilador01:=10;
			END_IF
			IF xDesligaFimVentilador01 THEN
				PassoVentilador01:=80;
			END_IF
			IF  xSemEnergia THEN
				PassoVentilador01:=80;
			END_IF
			IF NOT xVentPassHabilitado THEN
				PassoVentilador01:=80;
			END_IF
			IF xPause THEN
				PassoPauseVentilador01:=60;
				PassoVentilador01:=300;
			END_IF
			IF xAlarmeMotorVentilador01 THEN
				PassoAlmVentilador01:=60;
				PassoVentilador01:=400;
			END_IF

		80:	xPrimeiroEstagioVentilador01:=FALSE;
			xDesligaVentilador01:=FALSE;
			xDesligaFimVentilador01:=FALSE;
			xPrimeiroEstagioVentilador01:=FALSE;
			PassoVentilador01:=81;

		81:	xLigaMotorVentilador01:=FALSE;
			PassoVentilador01:=90;

		90:	PassoVentilador01:=91;

		91:PassoVentilador01:=0;

		// Emergência Pausa/Reinicio
		300:xLigaMotorVentilador01:=FALSE;
			PassoVentilador01:=301;

		301:PassoVentilador01:=302;

		302:IF xRestart THEN
				PassoVentilador01:=303;
			END_IF

		303:PassoVentilador01:=PassoPauseVentilador01;

		// Alarme Motor Parada/Reinicio
		400:xLigaMotorVentilador01:=FALSE;
			PassoVentilador01:=401;

		401:PassoVentilador01:=402;

		402:IF xRestart AND xInvVentilador01Habilitado THEN
				PassoVentilador01:=PassoAlmVentilador01;
			END_IF

END_CASE
// MOVIMENTAÇÃO PELO COMANDO ENTRADAS DIGITAIS DO INVERSOR
// Comando e Direção
xMotorVentilador01:=xLigaMotorVentilador01;

//InversorVentila01.i_xAvanco:=xMotorVentilador01;

// Velocidade
//InversorVentila01.i_iFreqRef:=iVelocidadeVentilador01;

// Velocidade
rVelocidadeVentilador01:=INT_TO_REAL(iVelocidadeVentilador01);
rVelocidadeVentilador01HZ:=((rVelocidadeVentilador01*600)/1800);
dVelocidadeVentilador01HZ:=REAL_TO_DINT(rVelocidadeVentilador01HZ);
iVelocidadeVentilador01HZ:=DINT_TO_INT(dVelocidadeVentilador01HZ);

iRefFreqVent01Pid:=iVelocidadeVentilador01HZ*10;

PIDVENT01.i_stPid.rLowLim:=0;
PIDVENT01.i_stPid.rHighLim:=100;
PIDVENT01.i_stPid.rTargCyclTime:=10;

PIDVENT01(
	i_xEn:= 		TRUE,
	i_rSp:= 		iRefFreqVent01Pid,
	i_rPv1:= 		iFrequenciaMotorVentilador01,
	i_iPv2:= 		,
	i_xHold:= 		,
	i_rKp:= 		10,//rGanhoPorporcionaKp,
	i_rTn:= 		0.8,//rGanhoIntegralKi,
	i_rTv:= 		2,//rGanhoDerivativoKd,
	i_rTd:= 		,
	i_xManMode:= 	,
	i_rManVal:= 	,
	i_stPid:= 		,
	i_xErrRst:= 	,
	q_xEn=> 		,
	q_xBusy=> 		,
	q_rPidOput=> 	rPidSaidaVent01,
	q_xMinLimActv=> ,
	q_xMaxLimActv=> ,
	q_xARWActv=> 	,
	q_xErr=> 		,
	q_uiErrId=> 	,
	q_sErrMsge=> 	,
	q_sFBstat=> 	);

//iAnaFreqRefVentilador01:=REAL_TO_INT (rPidSaidaVent01*17.0);

iAnaFreqRefVentilador01:=iRefFreqVent01Pid;
//------------------------------------------------------------------------\\
IF xOperacaoManual THEN
	PassoVentilador01:=0;
	PassoPauseVentilador01:=0;
	PassoAlmVentilador01:=0;
	xLigaVentilador01:=FALSE;
	xDesligaVentilador01:=FALSE;
	xDesligaFimVentilador01:=FALSE;
	xFimVentilacao01:=FALSE;
	xPrimeiroEstagioVentilador01:=FALSE;
	xVelocidadeVentilador01Ok:=FALSE;
	xFechaVenezVentPassV01:=FALSE;
	xLigaMotorVentilador01:=FALSE;
END_IF

IF iFrequenciaMotorVentilador01>=iVelocidade01Ventilador01 AND xPrimeiroEstagioVentilador01 THEN
	xVelocidadeVentilador01Ok:=TRUE;
END_IF

IF NOT xPrimeiroEstagioVentilador01 THEN
	xVelocidadeVentilador01Ok:=FALSE;
END_IF

(* ---- M_Ventilador02.prg.st ---- *)
PROGRAM M_Ventilador02
VAR
	PassoVentilador02: INT;
	PassoPauseVentilador02: INT;
	PassoAlmVentilador02: INT;
	PulsoLigaVentilador02: PulsoPositivo;
	/// Bloco Movimenta Guilhotina do Resfriador
	McMoveVelocityVentilador02: GIPLC.MC_MoveVelocity;
	/// Bloco Desliga Motor Guilhotina do Resfriador
	McStopVentilador02: GIPLC.MC_Stop;
	xExecutaMovVentilador02: BOOL;
	xExecutaStopVentilador02: BOOL;
	xStopVentilador02Done: BOOL;
	iVelocidadeVentilador02: INT;
	xLigaVentilador02: BOOL;
	xFimVentilacao02: BOOL;
	xLigaTempoVentilador02: BOOL;
	xPulsoLigaVentilador02: BOOL;
	xLigaVent02SairForno: BOOL;
	xTempoMvVent02In: BOOL;
	xTempoMvVent02Q: BOOL;
	TempoMvVent02: ton;
END_VAR

IF xEspessuraVidroFino THEN
	IF (iTempoAquecFornoRestante<=iTempoLigaVentilador02VidroFino) AND (iTempoAquecFornoRestante>0) AND xFornoEmCiclo THEN
		xLigaTempoVentilador02:=TRUE;
	ELSE
		xLigaTempoVentilador02:=FALSE;
	END_IF
ELSE
	IF (iTempoAquecFornoRestante<=iTempoLigaVentilador02VidroGros) AND (iTempoAquecFornoRestante>0) AND xFornoEmCiclo THEN
		xLigaTempoVentilador02:=TRUE;
	ELSE
		xLigaTempoVentilador02:=FALSE;
	END_IF
END_IF

xLigaVent02SairForno:=xSairForno AND xFornoEmCiclo AND xFornoComCarga;

PulsoLigaVentilador02(Entrada:= xLigaTempoVentilador02 OR xLigaVent02SairForno OR xLigaVent02FimForno, SaidaPulsoPo=>xPulsoLigaVentilador02 );
IF xPulsoLigaVentilador02 THEN
	xLigaVentilador02:=TRUE;
	xFechaVenezVentPassV02:=TRUE;//-> TASK/T_VenezianaVentInfPass
END_IF

(*IF xDesligaVentilador02 THEN
	xFimVentilacao02:=TRUE;
	xDesligaVentilador02:=FALSE;
END_IF*)

TempoMvVent02(IN:= xTempoMvVent02In, PT:=T#2S , Q=> xTempoMvVent02Q, ET=> );

// SEQUENCIA DE FUNCIONAMENTO

iVelocidade02Ventilador02:=iVelocidade01Ventilador02;
iVelocidade03Ventilador02:=iVelocidade01Ventilador02;

CASE PassoVentilador02 OF

		0:	IF xLigaVentilador02 THEN
				PassoVentilador02:=10;
			END_IF

		10:	xLigaVentilador02:=FALSE;
			xDesligaFimVentilador02:=FALSE;
			xPrimeiroEstagioVentilador02:=TRUE;
			xSegundoEstagioVentilador02:=FALSE;
			xTerceiroEstagioVentilador02:=FALSE;
			PassoVentilador02:=15;

		15:	PassoVentilador02:=16;

		16:	IF  xSemEnergia THEN
				PassoVentilador02:=80;
			ELSIF xPause THEN
				PassoPauseVentilador02:=16;
				PassoVentilador02:=300;
			ELSIF xAlarmeMotorVentilador02 THEN
				PassoAlmVentilador02:=16;
				PassoVentilador02:=400;
			ELSE
				PassoVentilador02:=20;
			END_IF

		20:	iVelocidadeVentilador02:=iVelocidade01Ventilador02;
			PassoVentilador02:=21;

		21:	xExecutaMovVentilador02:=TRUE;
			PassoVentilador02:=22;

		22:	IF McMoveVelocityVentilador02.Busy THEN
				PassoVentilador02:=29;
			ELSE
				PassoVentilador02:=23;
			END_IF

		23:xExecutaMovVentilador02:=FALSE;
			xTempoMvVent02In:=TRUE;
			IF	xTempoMvVent02Q THEN
				PassoVentilador02:=24;
			END_IF

		24:	xTempoMvVent02In:=FALSE;
			xExecutaStopVentilador02:=TRUE;
			PassoVentilador02:=25;

		25:	xExecutaStopVentilador02:=FALSE;
			PassoVentilador02:=16;

		29:	xExecutaMovVentilador02:=FALSE;
			PassoVentilador02:=59;//30; (* Alterado Ventilador tempera passagem*)
		// Fica Parado no passo 30 aguardando o inicio do segundo Estágio
		30:	IF iVelocidadeVentilador02<>iVelocidade01Ventilador02 THEN
				PassoVentilador02:=20;
			END_IF
			IF xSegundoEstagioVentilador02 THEN //<-TASK/EstagiosResfriador
				PassoVentilador02:=40;
			END_IF
			IF xDesligaVentilador02 THEN
				PassoVentilador02:=41;
			END_IF
			IF  xSemEnergia THEN
				PassoVentilador02:=80;
			END_IF
			IF xPause THEN
				PassoPauseVentilador02:=20;
				PassoVentilador02:=300;
			END_IF
			IF xAlarmeMotorVentilador02 THEN
				PassoAlmVentilador02:=20;
				PassoVentilador02:=400;
			END_IF

		40:	xSegundoEstagioVentilador02:=FALSE;
			xDesligaVentilador02:=FALSE; // Zera memoria desliga vent caso esteja em 1
			PassoVentilador02:=41;

		41:	xPrimeiroEstagioVentilador02:=FALSE;
			iVelocidadeVentilador02:=iVelocidade02Ventilador02;
			PassoVentilador02:=42;

		42:	xExecutaMovVentilador02:=TRUE;
			PassoVentilador02:=43;

		43:	IF McMoveVelocityVentilador02.Busy THEN
				PassoVentilador02:=44;
			END_IF

		44:	xExecutaMovVentilador02:=FALSE;
			PassoVentilador02:=50;
		// Fica Parado no Passo 50 aguardando o inicio do Terceiro Estágio
		50:	IF iVelocidadeVentilador02<>iVelocidade02Ventilador02 THEN
				PassoVentilador02:=41;
			END_IF
			IF xTerceiroEstagioVentilador02 THEN //<-TASK/EstagiosResfriador
				PassoVentilador02:=51;
			END_IF
			IF xDesligaVentilador02 THEN
				PassoVentilador02:=52;
			END_IF
			IF  xSemEnergia THEN
				PassoVentilador02:=80;
			END_IF
			IF xPause THEN
				PassoPauseVentilador02:=41;
				PassoVentilador02:=300;
			END_IF
			IF xAlarmeMotorVentilador02 THEN
				PassoAlmVentilador02:=41;
				PassoVentilador02:=400;
			END_IF

		51:	xTerceiroEstagioVentilador02:=FALSE;
			xDesligaVentilador02:=FALSE; // Zera memoria desliga vent caso esteja em 1
			PassoVentilador02:=52;

		52:	xSegundoEstagioVentilador02:=FALSE;
			iVelocidadeVentilador02:=iVelocidade03Ventilador02;
			PassoVentilador02:=53;

		53:	xExecutaMovVentilador02:=TRUE;
			PassoVentilador02:=54;

		54:	IF McMoveVelocityVentilador02.Busy THEN
				PassoVentilador02:=55;
			END_IF

		55:	xExecutaMovVentilador02:=FALSE;
			PassoVentilador02:=59;

			// Fica Parado no Passo 59 Aguardando
		59:	IF iVelocidadeVentilador02<>iVelocidade03Ventilador02 THEN
				PassoVentilador02:=20;//52; (* Alterador Tempera de passagem *)
			END_IF
			IF xLigaVentilador02 THEN
				PassoVentilador02:=10;
			END_IF
			IF xDesligaVentilador02 AND NOT xFornoEmEspera THEN
				PassoVentilador02:=60;
			END_IF
			IF xDesligaVentilador02 AND xFornoEmEspera THEN
				PassoVentilador02:=80;
			END_IF
			IF  xSemEnergia THEN
				PassoVentilador02:=80;
			END_IF
			IF xPause THEN
				PassoPauseVentilador02:=20;//52; (* Alterador Tempera de passagem *)
				PassoVentilador02:=300;
			END_IF
			IF xAlarmeMotorVentilador02 THEN
				PassoAlmVentilador02:=20;//52; (* Alterador Tempera de passagem *)
				PassoVentilador02:=400;
			END_IF

		60:	xDesligaVentilador02:=FALSE;
			PassoVentilador02:=61;

		61:	iVelocidadeVentilador02:=iVelocidadeStbVent02Pass;//iVelocidadeStbVentilador02;
			PassoVentilador02:=62;

		62:	xExecutaMovVentilador02:=TRUE;
			PassoVentilador02:=63;

		63:	IF McMoveVelocityVentilador02.Busy THEN
				PassoVentilador02:=70;
			ELSE
				PassoVentilador02:=64;
			END_IF

		64:xExecutaMovVentilador02:=FALSE;
			xTempoMvVent02In:=TRUE;
			IF	xTempoMvVent02Q THEN
				PassoVentilador02:=65;
			END_IF

		65:	xTempoMvVent02In:=FALSE;
			xExecutaStopVentilador02:=TRUE;
			PassoVentilador02:=66;

		66:	xExecutaStopVentilador02:=FALSE;
			PassoVentilador02:=60;

		70:	xExecutaMovVentilador02:=FALSE;
			PassoVentilador02:=71;

		71:	IF iVelocidadeVentilador02<>iVelocidadeStbVent02Pass(*iVelocidadeStbVentilador02*) THEN
				PassoVentilador02:=61;
			END_IF
			IF xLigaVentilador02 THEN
				PassoVentilador02:=10;
			END_IF
			IF xDesligaFimVentilador02 THEN
				PassoVentilador02:=80;
			END_IF
			IF  xSemEnergia THEN
				PassoVentilador02:=80;
			END_IF
			IF xPause THEN
				PassoPauseVentilador02:=60;
				PassoVentilador02:=300;
			END_IF
			IF xAlarmeMotorVentilador02 THEN
				PassoAlmVentilador02:=60;
				PassoVentilador02:=400;
			END_IF

		80:	xPrimeiroEstagioVentilador02:=FALSE;
			xDesligaVentilador02:=FALSE;
			xDesligaFimVentilador02:=FALSE;
			xExecutaStopVentilador02:=TRUE;
			PassoVentilador02:=81;

		81:	IF	xStopVentilador02Done THEN
				PassoVentilador02:=90;
			END_IF

		90:	xExecutaStopVentilador02:=FALSE;
			PassoVentilador02:=91;

		91:PassoVentilador02:=0;

		// Emergência Pausa/Reinicio
		300:xExecutaStopVentilador02:=TRUE;
			PassoVentilador02:=301;

		301:xExecutaMovVentilador02:=FALSE;
			xExecutaStopVentilador02:=FALSE;
			PassoVentilador02:=302;

		302:IF xRestart THEN
				PassoVentilador02:=303;
			END_IF

		303:IF xInvVentilador02Habilitado THEN
				PassoVentilador02:=PassoPauseVentilador02;
			END_IF

		// Alarme Motor Parada/Reinicio
		400:xExecutaStopVentilador02:=TRUE;
			PassoVentilador02:=401;

		401:xExecutaStopVentilador02:=FALSE;
			xExecutaMovVentilador02:=FALSE;
			PassoVentilador02:=402;

		402:IF xRestart AND xInvVentilador02Habilitado THEN
				PassoVentilador02:=PassoAlmVentilador02;
			END_IF

END_CASE

// BLOCOS DE EXECUÇÃO CANOPEN
//McMoveVelocityVentilador02(Execute:= xExecutaMovVentilador02,	Velocity:=iVelocidadeVentilador02,	Axis:= Ventilador_02,	InVelocity=> ,	Busy=> ,CommandAborted=> , Error=> );
//McStopVentilador02(Execute:=xExecutaStopVentilador02,	Axis:= Ventilador_02, Done=>xStopVentilador02Done ,Busy=> , Error=> );

IF xOperacaoManual THEN
	PassoVentilador02:=0;
	PassoPauseVentilador02:=0;
	PassoAlmVentilador02:=0;
	xExecutaMovVentilador02:=FALSE;
	xExecutaStopVentilador02:=FALSE;
	xLigaVentilador02:=FALSE;
	xDesligaVentilador02:=FALSE;
	xDesligaFimVentilador02:=FALSE;
	xFimVentilacao02:=FALSE;
	xPrimeiroEstagioVentilador02:=FALSE;
	xVelocidadeVentilador02Ok:=FALSE;
	xFechaVenezVentPassV02:=FALSE;
END_IF

IF  xEmergencia THEN
	xExecutaStopVentilador02:=TRUE;
	xExecutaMovVentilador02:=FALSE;
ELSE
	xExecutaStopVentilador02:=FALSE;
END_IF

IF iFrequenciaMotorVentilador02>=iVelocidade01Ventilador02 AND xPrimeiroEstagioVentilador02 THEN
	xVelocidadeVentilador02Ok:=TRUE;
END_IF

IF NOT xPrimeiroEstagioVentilador02 THEN
	xVelocidadeVentilador02Ok:=FALSE;
END_IF

(* ---- M_Ventilador03.prg.st ---- *)
PROGRAM M_Ventilador03
VAR
	PassoVentilador03: INT;
	PassoPauseVentilador03: INT;
	PassoAlmVentilador03: INT;
	PulsoLigaVentilador03: PulsoPositivo;
	iVelocidadeVentilador03: INT;
	xLigaVentilador03: BOOL;
	xFimVentilacao03: BOOL;
	xLigaTempoVentilador03: BOOL;
	xPulsoLigaVentilador03: BOOL;
	xLigaVent03SairForno: BOOL;
	xTempoMvVent03In: BOOL;
	xTempoMvVent03Q: BOOL;
	TempoMvVent03: ton;
	xLigaMotorVentilador03: BOOL;
	iVelocidadeVentilador03HZ: INT;
	dVelocidadeVentilador03HZ: DINT;
	rVelocidadeVentilador03HZ:REAL;
	rVelocidadeVentilador03 :REAL;
END_VAR

IF xEspessuraVidroFino THEN
	IF (iTempoAquecFornoRestante<=iTempoLigaVentilador03VidroFino) AND (iTempoAquecFornoRestante>0) AND xFornoEmCiclo THEN
		xLigaTempoVentilador03:=TRUE;
	ELSE
		xLigaTempoVentilador03:=FALSE;
	END_IF
ELSE
	IF (iTempoAquecFornoRestante<=iTempoLigaVentilador03VidroGros) AND (iTempoAquecFornoRestante>0) AND xFornoEmCiclo THEN
		xLigaTempoVentilador03:=TRUE;
	ELSE
		xLigaTempoVentilador03:=FALSE;
	END_IF
END_IF

xLigaVent03SairForno:=xSairForno AND xFornoEmCiclo AND xFornoComCarga;

PulsoLigaVentilador03(Entrada:= xLigaTempoVentilador03 OR xLigaVent03SairForno OR xLigaVent03FimForno, SaidaPulsoPo=>xPulsoLigaVentilador03 );
IF xPulsoLigaVentilador03 THEN
	xLigaVentilador03:=TRUE;
	xReajustaAlturaDuctosSup02:=TRUE;
	xReajustaAlturaDuctosInf02:=TRUE;
END_IF

TempoMvVent03(IN:= xTempoMvVent03In, PT:=T#2S , Q=> xTempoMvVent03Q, ET=> );

// SEQUENCIA DE FUNCIONAMENTO

CASE PassoVentilador03 OF

		0:	IF xLigaVentilador03 THEN
				IF xResfriadorCarregado THEN
					PassoVentilador03:=2;
				ELSE
					PassoVentilador03:=10;
				END_IF
			END_IF

		2: IF NOT xResfriadorCarregado THEN
				PassoVentilador03:=10;
		   END_IF

		10:	xLigaVentilador03:=FALSE;
			xDesligaVentilador03:=FALSE;
			xDesligaFimVentilador03:=FALSE;
			xSegundoEstagioVentilador03:=FALSE;
			xTerceiroEstagioVentilador03:=FALSE;
			PassoVentilador03:=15;

		15:	xPrimeiroEstagioVentilador03:=TRUE;
			PassoVentilador03:=16;

		16:	IF  xSemEnergia THEN
				PassoVentilador03:=80;
			ELSIF xPause THEN
				PassoPauseVentilador03:=16;
				PassoVentilador03:=300;
			ELSIF xAlarmeMotorVentilador03 THEN
				PassoAlmVentilador03:=16;
				PassoVentilador03:=400;
			ELSE
				PassoVentilador03:=20;
			END_IF

		20:	iVelocidadeVentilador03:=REAL_TO_INT(iVelocidade01Ventilador03);
			PassoVentilador03:=21;

		21:	xLigaMotorVentilador03:=TRUE;
			PassoVentilador03:=22;

		22:	PassoVentilador03:=29;

		29:	PassoVentilador03:=30;

		// Fica Parado no passo 30 aguardando o inicio do segundo Estágio
		30:	IF iVelocidadeVentilador03<>REAL_TO_INT(iVelocidade01Ventilador03) THEN
				PassoVentilador03:=20;
			END_IF
			IF xSegundoEstagioVentilador03 THEN //<-TASK/EstagiosResfriador
				PassoVentilador03:=40;
			END_IF
			IF xLigaVentilador03 THEN
				PassoVentilador03:=10;
			END_IF
			IF xDesligaVentilador03 AND NOT xPrimeiroEstagioVentilador03 THEN
				PassoVentilador03:=41;
			END_IF
			IF  xSemEnergia THEN
				PassoVentilador03:=80;
			END_IF
			IF xPause THEN
				PassoPauseVentilador03:=20;
				PassoVentilador03:=300;
			END_IF
			IF xAlarmeMotorVentilador03 THEN
				PassoAlmVentilador03:=20;
				PassoVentilador03:=400;
			END_IF

		40:	xSegundoEstagioVentilador03:=FALSE;
			xDesligaVentilador03:=FALSE; // Zera memoria desliga vent caso esteja em 1
			PassoVentilador03:=42;

		41:	xLigaMotorVentilador03:=TRUE;
			PassoVentilador03:=42;

		42:	xPrimeiroEstagioVentilador03:=FALSE;
			iVelocidadeVentilador03:=REAL_TO_INT(iVelocidade02Ventilador03);
			PassoVentilador03:=43;

		43:	PassoVentilador03:=44;

		44:	PassoVentilador03:=50;
		// Fica Parado no Passo 50 aguardando o inicio do Terceiro Estágio
		50:	IF iVelocidadeVentilador03<>REAL_TO_INT(iVelocidade02Ventilador03) THEN
				PassoVentilador03:=41;
			END_IF
			IF xTerceiroEstagioVentilador03 THEN //<-TASK/EstagiosResfriador
				PassoVentilador03:=51;
			END_IF
			IF xLigaVentilador03 THEN
				PassoVentilador03:=10;
			END_IF
			IF xDesligaVentilador03 THEN
				PassoVentilador03:=52;
			END_IF
			IF  xSemEnergia THEN
				PassoVentilador03:=80;
			END_IF
			IF xPause THEN
				PassoPauseVentilador03:=41;
				PassoVentilador03:=300;
			END_IF
			IF xAlarmeMotorVentilador03 THEN
				PassoAlmVentilador03:=41;
				PassoVentilador03:=400;
			END_IF

		51:	xTerceiroEstagioVentilador03:=FALSE;
			xDesligaVentilador03:=FALSE; // Zera memoria desliga vent caso esteja em 1
			PassoVentilador03:=53;

		52:	xLigaMotorVentilador03:=TRUE;
			PassoVentilador03:=53;

		53:	xSegundoEstagioVentilador03:=FALSE;
			iVelocidadeVentilador03:=REAL_TO_INT(iVelocidade03Ventilador03);
			PassoVentilador03:=54;

		54:	PassoVentilador03:=55;

		55:	PassoVentilador03:=59;

			// Fica Parado no Passo 59 Aguardando
		59:	IF iVelocidadeVentilador03<>REAL_TO_INT(iVelocidade03Ventilador03) THEN
				PassoVentilador03:=52;
			END_IF
			IF xLigaVentilador03 THEN
				PassoVentilador03:=10;
			END_IF
			IF xDesligaVentilador03 AND NOT xFornoEmEspera THEN
				PassoVentilador03:=60;
			END_IF
			IF xDesligaVentilador03 AND xFornoEmEspera THEN
				PassoVentilador03:=80;
			END_IF
			IF  xSemEnergia THEN
				PassoVentilador03:=80;
			END_IF
			IF xPause THEN
				PassoPauseVentilador03:=52;
				PassoVentilador03:=300;
			END_IF
			IF xAlarmeMotorVentilador03 THEN
				PassoAlmVentilador03:=52;
				PassoVentilador03:=400;
			END_IF

		60:	xDesligaVentilador03:=FALSE;
			PassoVentilador03:=62;

		61:	IF iVelocidadeStbVentilador03<>0 THEN
				PassoVentilador03:=62;
			ELSE
				PassoVentilador03:=63;
			END_IF

		62:	xLigaMotorVentilador03:=TRUE;
			PassoVentilador03:=70;

		63:	xLigaMotorVentilador03:=FALSE;
			PassoVentilador03:=70;

		70:	iVelocidadeVentilador03:=iVelocidadeStbVentilador03;
			PassoVentilador03:=71;

		71:	IF iVelocidadeVentilador03<>iVelocidadeStbVentilador03 THEN
				PassoVentilador03:=61;
			END_IF
			IF xLigaVentilador03 THEN
				PassoVentilador03:=10;
			END_IF
			IF xDesligaFimVentilador03 THEN
				PassoVentilador03:=80;
			END_IF
			IF  xSemEnergia THEN
				PassoVentilador03:=80;
			END_IF
			IF xPause THEN
				PassoPauseVentilador03:=61;
				PassoVentilador03:=300;
			END_IF
			IF xAlarmeMotorVentilador03 THEN
				PassoAlmVentilador03:=61;
				PassoVentilador03:=400;
			END_IF

		80:	xPrimeiroEstagioVentilador03:=FALSE;
			xDesligaVentilador03:=FALSE;
			xDesligaFimVentilador03:=FALSE;
			PassoVentilador03:=81;

		81:	xLigaMotorVentilador03:=FALSE;
			PassoVentilador03:=90;

		90: PassoVentilador03:=91;

		91:PassoVentilador03:=0;

		// Emergência Pausa/Reinicio
		300:xLigaMotorVentilador03:=FALSE;
			PassoVentilador03:=301;

		301:PassoVentilador03:=302;

		302:IF xRestart THEN
				PassoVentilador03:=303;
			END_IF

		303:PassoVentilador03:=PassoPauseVentilador03;

		// Alarme Motor Parada/Reinicio
		400:xLigaMotorVentilador03:=FALSE;
			PassoVentilador03:=401;

		401:PassoVentilador03:=402;

		402:IF xRestart AND iCanOpenInverVentila03StateOk THEN
				PassoVentilador03:=PassoAlmVentilador03;
			END_IF

END_CASE
// MOVIMENTAÇÃO PELO COMANDO ENTRADAS DIGITAIS DO INVERSOR
// Comando e Direção
xMotorVentilador03:=xLigaMotorVentilador03;

InversorVentila03.i_xAvanco:=xMotorVentilador03;

// Velocidade
rVelocidadeVentilador03:=INT_TO_REAL(iVelocidadeVentilador03);
rVelocidadeVentilador03HZ:=((rVelocidadeVentilador03*600)/1787);
dVelocidadeVentilador03HZ:=REAL_TO_DINT(rVelocidadeVentilador03HZ);
iVelocidadeVentilador03HZ:=DINT_TO_INT(dVelocidadeVentilador03HZ);

InversorVentila03.i_iFreqRef:=iVelocidadeVentilador03HZ;

//InversorVentila03.i_iFreqRef:=iVelocidadeVentilador03;
//------------------------------------------------------------------------\\
IF xOperacaoManual THEN
	PassoVentilador03:=0;
	PassoPauseVentilador03:=0;
	PassoAlmVentilador03:=0;
	xLigaVentilador03:=FALSE;
	xDesligaVentilador03:=FALSE;
	xDesligaFimVentilador03:=FALSE;
	xFimVentilacao03:=FALSE;
	xPrimeiroEstagioVentilador03:=FALSE;
	xVelocidadeVentilador03Ok:=FALSE;
	xTempoMvVent03In:=FALSE;
	xLigaMotorVentilador03:=FALSE;
END_IF

IF iFrequenciaMotorVentilador03>=REAL_TO_INT(iVelocidade01Ventilador03/100) AND xPrimeiroEstagioVentilador03 THEN
	xVelocidadeVentilador03Ok:=TRUE;
END_IF

IF NOT xPrimeiroEstagioVentilador03 THEN
	xVelocidadeVentilador03Ok:=FALSE;
END_IF

(* ---- M_Ventilador04.prg.st ---- *)
PROGRAM M_Ventilador04
VAR
	PassoVentilador04: INT;
	PassoPauseVentilador04: INT;
	PassoAlmVentilador04: INT;
	PulsoLigaVentilador04: PulsoPositivo;
	/// Bloco Movimenta Guilhotina do Resfriador
	McMoveVelocityVentilador04: GIPLC.MC_MoveVelocity;
	/// Bloco Desliga Motor Guilhotina do Resfriador
	McStopVentilador04: GIPLC.MC_Stop;
	xExecutaMovVentilador04: BOOL;
	xExecutaStopVentilador04: BOOL;
	xStopVentilador04Done: BOOL;
	iVelocidadeVentilador04: INT;
	xLigaVentilador04: BOOL;
	xFimVentilacao04: BOOL;
	xLigaTempoVentilador04: BOOL;
	xPulsoLigaVentilador04: BOOL;
	xLigaVent04SairForno: BOOL;
	xTempoMvVent04In: BOOL;
	xTempoMvVent04Q: BOOL;
	TempoMvVent04: ton;
END_VAR

IF xEspessuraVidroFino THEN
	IF (iTempoAquecFornoRestante<=iTempoLigaVentilador04VidroFino) AND (iTempoAquecFornoRestante>0) AND xFornoEmCiclo THEN
		xLigaTempoVentilador04:=TRUE;
	ELSE
		xLigaTempoVentilador04:=FALSE;
	END_IF
ELSE
	IF (iTempoAquecFornoRestante<=iTempoLigaVentilador04VidroGros) AND (iTempoAquecFornoRestante>0) AND xFornoEmCiclo THEN
		xLigaTempoVentilador04:=TRUE;
	ELSE
		xLigaTempoVentilador04:=FALSE;
	END_IF
END_IF

xLigaVent04SairForno:=xSairForno AND xFornoEmCiclo AND xFornoComCarga;

PulsoLigaVentilador04(Entrada:= xLigaTempoVentilador04 OR xLigaVent04SairForno OR xLigaVent04FimForno, SaidaPulsoPo=>xPulsoLigaVentilador04 );
IF xPulsoLigaVentilador04 THEN
	xLigaVentilador04:=TRUE;
END_IF

TempoMvVent04(IN:= xTempoMvVent04In, PT:=T#2S , Q=> xTempoMvVent04Q, ET=> );

// SEQUENCIA DE FUNCIONAMENTO

CASE PassoVentilador04 OF

		0:	IF xLigaVentilador04 THEN
				IF xResfriadorCarregado THEN
					PassoVentilador04:=2;
				ELSE
					PassoVentilador04:=10;
				END_IF
			END_IF

		2: IF NOT xResfriadorCarregado THEN
				PassoVentilador04:=10;
		   END_IF

		10:	xLigaVentilador04:=FALSE;
			xDesligaVentilador04:=FALSE;
			xDesligaFimVentilador04:=FALSE;
			xSegundoEstagioVentilador04:=FALSE;
			xTerceiroEstagioVentilador04:=FALSE;
			PassoVentilador04:=15;

		15:	xPrimeiroEstagioVentilador04:=TRUE;
			PassoVentilador04:=16;

		16:	IF  xSemEnergia THEN
				PassoVentilador04:=80;
			ELSIF xPause THEN
				PassoPauseVentilador04:=16;
				PassoVentilador04:=300;
			ELSIF xAlarmeMotorVentilador04 THEN
				PassoAlmVentilador04:=16;
				PassoVentilador04:=400;
			ELSE
				PassoVentilador04:=20;
			END_IF

		20:	iVelocidadeVentilador04:=iVelocidade01Ventilador04;
			PassoVentilador04:=21;

		21:	xExecutaMovVentilador04:=TRUE;
			PassoVentilador04:=22;

		22:	IF McMoveVelocityVentilador04.Busy THEN
				PassoVentilador04:=29;
			ELSE
				PassoVentilador04:=23;
			END_IF

		23:xExecutaMovVentilador04:=FALSE;
			xTempoMvVent04In:=TRUE;
			IF	xTempoMvVent04Q THEN
				PassoVentilador04:=24;
			END_IF

		24:	xTempoMvVent04In:=FALSE;
			xExecutaStopVentilador04:=TRUE;
			PassoVentilador04:=25;

		25:	xExecutaStopVentilador04:=FALSE;
			PassoVentilador04:=16;

		29:	xExecutaMovVentilador04:=FALSE;
			PassoVentilador04:=30;
		// Fica Parado no passo 30 aguardando o inicio do segundo Estágio
		30:	IF iVelocidadeVentilador04<>iVelocidade01Ventilador04 THEN
				PassoVentilador04:=20;
			END_IF
			IF xSegundoEstagioVentilador04 THEN //<-TASK/EstagiosResfriador
				PassoVentilador04:=40;
			END_IF
			IF xDesligaVentilador04 THEN
				PassoVentilador04:=41;
			END_IF
			IF  xSemEnergia THEN
				PassoVentilador04:=80;
			END_IF
			IF xPause THEN
				PassoPauseVentilador04:=20;
				PassoVentilador04:=300;
			END_IF
			IF xAlarmeMotorVentilador04 THEN
				PassoAlmVentilador04:=20;
				PassoVentilador04:=400;
			END_IF

		40:	xSegundoEstagioVentilador04:=FALSE;
			xDesligaVentilador04:=FALSE; // Zera memoria desliga vent caso esteja em 1
			PassoVentilador04:=41;

		41:	xPrimeiroEstagioVentilador04:=FALSE;
			iVelocidadeVentilador04:=iVelocidade02Ventilador04;
			PassoVentilador04:=42;

		42:	xExecutaMovVentilador04:=TRUE;
			PassoVentilador04:=43;

		43:	IF McMoveVelocityVentilador04.Busy THEN
				PassoVentilador04:=44;
			ELSE
				PassoVentilador04:=45;
			END_IF

		45:xExecutaMovVentilador04:=FALSE;
			xTempoMvVent04In:=TRUE;
			IF	xTempoMvVent04Q THEN
				PassoVentilador04:=46;
			END_IF

		46:	xTempoMvVent04In:=FALSE;
			xExecutaStopVentilador04:=TRUE;
			PassoVentilador04:=47;

		47:	xExecutaStopVentilador04:=FALSE;
			PassoVentilador04:=41;

		44:	xExecutaMovVentilador04:=FALSE;
			PassoVentilador04:=50;
		// Fica Parado no Passo 50 aguardando o inicio do Terceiro Estágio
		50:	IF iVelocidadeVentilador04<>iVelocidade02Ventilador04 THEN
				PassoVentilador04:=41;
			END_IF
			IF xTerceiroEstagioVentilador04 THEN //<-TASK/EstagiosResfriador
				PassoVentilador04:=51;
			END_IF
			IF xDesligaVentilador04 THEN
				PassoVentilador04:=52;
			END_IF
			IF  xSemEnergia THEN
				PassoVentilador04:=80;
			END_IF
			IF xPause THEN
				PassoPauseVentilador04:=41;
				PassoVentilador04:=300;
			END_IF
			IF xAlarmeMotorVentilador04 THEN
				PassoAlmVentilador04:=41;
				PassoVentilador04:=400;
			END_IF

		51:	xTerceiroEstagioVentilador04:=FALSE;
			xDesligaVentilador04:=FALSE; // Zera memoria desliga vent caso esteja em 1
			PassoVentilador04:=52;

		52:	xSegundoEstagioVentilador04:=FALSE;
			iVelocidadeVentilador04:=iVelocidade03Ventilador04;
			PassoVentilador04:=53;

		53:	xExecutaMovVentilador04:=TRUE;
			PassoVentilador04:=54;

		54:	IF McMoveVelocityVentilador04.Busy THEN
				PassoVentilador04:=55;
			ELSE
				PassoVentilador04:=56;
			END_IF

		56:xExecutaMovVentilador04:=FALSE;
			xTempoMvVent04In:=TRUE;
			IF	xTempoMvVent04Q THEN
				PassoVentilador04:=57;
			END_IF

		57:	xTempoMvVent04In:=FALSE;
			xExecutaStopVentilador04:=TRUE;
			PassoVentilador04:=58;

		58:	xExecutaStopVentilador04:=FALSE;
			PassoVentilador04:=52;

		55:	xExecutaMovVentilador04:=FALSE;
			PassoVentilador04:=59;

			// Fica Parado no Passo 59 Aguardando
		59:	IF iVelocidadeVentilador04<>iVelocidade03Ventilador04 THEN
				PassoVentilador04:=52;
			END_IF
			IF xLigaVentilador04 THEN
				PassoVentilador04:=10;
			END_IF
			IF xDesligaVentilador04 AND NOT xFornoEmEspera THEN
				PassoVentilador04:=60;
			END_IF
			IF xDesligaVentilador04 AND xFornoEmEspera THEN
				PassoVentilador04:=80;
			END_IF
			IF  xSemEnergia THEN
				PassoVentilador04:=80;
			END_IF
			IF xPause THEN
				PassoPauseVentilador04:=52;
				PassoVentilador04:=300;
			END_IF
			IF xAlarmeMotorVentilador04 THEN
				PassoAlmVentilador04:=52;
				PassoVentilador04:=400;
			END_IF

		60:	xDesligaVentilador04:=FALSE;
			PassoVentilador04:=61;

		61:	iVelocidadeVentilador04:=iVelocidadeStbVentilador04;
			PassoVentilador04:=62;

		62:	xExecutaMovVentilador04:=TRUE;
			PassoVentilador04:=63;

		63:	IF McMoveVelocityVentilador04.Busy THEN
				PassoVentilador04:=70;
			ELSE
				PassoVentilador04:=64;
			END_IF

		64:xExecutaMovVentilador04:=FALSE;
			xTempoMvVent04In:=TRUE;
			IF	xTempoMvVent04Q THEN
				PassoVentilador04:=65;
			END_IF

		65:	xTempoMvVent04In:=FALSE;
			xExecutaStopVentilador04:=TRUE;
			PassoVentilador04:=66;

		66:	xExecutaStopVentilador04:=FALSE;
			PassoVentilador04:=60;

		70:	xExecutaMovVentilador04:=FALSE;
			PassoVentilador04:=71;

		71:	IF iVelocidadeVentilador04<>iVelocidadeStbVentilador04 THEN
				PassoVentilador04:=61;
			END_IF
			IF xLigaVentilador04 THEN
				PassoVentilador04:=10;
			END_IF
			IF xDesligaFimVentilador04 THEN
				PassoVentilador04:=80;
			END_IF
			IF  xSemEnergia THEN
				PassoVentilador04:=80;
			END_IF
			IF xPause THEN
				PassoPauseVentilador04:=60;
				PassoVentilador04:=300;
			END_IF
			IF xAlarmeMotorVentilador04 THEN
				PassoAlmVentilador04:=60;
				PassoVentilador04:=400;
			END_IF

		80:	xPrimeiroEstagioVentilador04:=FALSE;
			xDesligaVentilador04:=FALSE;
			xDesligaFimVentilador04:=FALSE;
			xExecutaStopVentilador04:=TRUE;
			PassoVentilador04:=81;

		81:	IF	xStopVentilador04Done THEN
				PassoVentilador04:=90;
			END_IF

		90:	xExecutaStopVentilador04:=FALSE;
			PassoVentilador04:=91;

		91:PassoVentilador04:=0;

		// Emergência Pausa/Reinicio
		300:xExecutaStopVentilador04:=TRUE;
			PassoVentilador04:=301;

		301:xExecutaMovVentilador04:=FALSE;
			xExecutaStopVentilador04:=FALSE;
			PassoVentilador04:=302;

		302:IF xRestart THEN
				PassoVentilador04:=303;
			END_IF

		303:IF xInvVentilador04Habilitado THEN
				PassoVentilador04:=PassoPauseVentilador04;
			END_IF

		// Alarme Motor Parada/Reinicio
		400:xExecutaStopVentilador04:=TRUE;
			PassoVentilador04:=401;

		401:xExecutaStopVentilador04:=FALSE;
			xExecutaMovVentilador04:=FALSE;
			PassoVentilador04:=402;

		402:IF xRestart AND xInvVentilador04Habilitado THEN
				PassoVentilador04:=PassoAlmVentilador04;
			END_IF

END_CASE

// BLOCOS DE EXECUÇÃO CANOPEN
//McMoveVelocityVentilador04(Execute:= xExecutaMovVentilador04,	Velocity:=iVelocidadeVentilador04,	Axis:= Ventilador_04,	InVelocity=> ,	Busy=> ,CommandAborted=> , Error=> );
//McStopVentilador04(Execute:=xExecutaStopVentilador04,	Axis:= Ventilador_04, Done=>xStopVentilador04Done ,Busy=> , Error=> );

IF xOperacaoManual THEN
	PassoVentilador04:=0;
	PassoPauseVentilador04:=0;
	PassoAlmVentilador04:=0;
	xExecutaMovVentilador04:=FALSE;
	xExecutaStopVentilador04:=FALSE;
	xLigaVentilador04:=FALSE;
	xDesligaVentilador04:=FALSE;
	xDesligaFimVentilador04:=FALSE;
	xFimVentilacao04:=FALSE;
	xPrimeiroEstagioVentilador04:=FALSE;
	xVelocidadeVentilador04Ok:=FALSE;
	xTempoMvVent04In:=FALSE;
END_IF

//IF  xEmergencia THEN
//	xExecutaStopVentilador04:=TRUE;
//	xExecutaMovVentilador04:=FALSE;
//ELSE
//	xExecutaStopVentilador04:=FALSE;
//END_IF

IF iFrequenciaMotorVentilador04>=iVelocidade01Ventilador04 AND xPrimeiroEstagioVentilador04 THEN
	xVelocidadeVentilador04Ok:=TRUE;
END_IF

IF NOT xPrimeiroEstagioVentilador04 THEN
	xVelocidadeVentilador04Ok:=FALSE;
END_IF

(* ---- N_Grades.prg.st ---- *)
PROGRAM N_Grades
VAR
	GradeEntrada: Grade;
	GradeSaida: Grade;
	TpBtGradEnt: TP;
	xTpBtGradEntIn: BOOL;
	xTpBtGradEntQ: BOOL;
	xDesabGradeEntrada: BOOL;
	xHabilGradeEntrada: BOOL;
END_VAR

// Grade Mesa de Entrada

xDesabGradeEntrada:= xCarregandoForno OR xRetornandoForno;
xHabilGradeEntrada:= NOT xDesabGradeEntrada;

GradeEntrada(
	LigaDesl:= xBtGradeEntrada,
	Libera:= TRUE,//xS01PistPneumRecuado AND xS03PistHidraulRecuado,
	Liga:= ,
	Desl:= xDesabGradeEntrada,//xMotorEntradaLigado,
	Alarme01:=,// xEmergencia,
	StatusSaida=> xValvulaGradeEntrada);

//Grade Mesa de Saída
GradeSaida(
	LigaDesl:= xBtGradeSaida,
	Libera:=TRUE,
	Liga:= ,
	Desl:= xDesceGradeMesaSaida OR xMotorSaidaLigado,
	Alarme01:= xEmergencia,
	StatusSaida=> xValvulaGradeSaida);

IF xDesceGradeMesaSaida THEN
	xDesceGradeMesaSaida:=FALSE;
END_IF

//IF xOperacaoManual THEN
//	xDesceGradeMesaSaida:=TRUE;
//END_IF;

(* ---- N_MesaBasculante.prg.st ---- *)
PROGRAM N_MesaBasculante
VAR
	PassoMesaBasculEnt: INT;
	PassoPauseBasculEnt: INT;
	PassoAlmBasculEnt: INT;
	TonAbreBraco: TON;
	TonAbreBracoIn: BOOL;
	TonAbreBracoQ: BOOL;
	TonFechaBraco: TON;
	TonFechaBracoIn: BOOL;
	TonFechaBracoQ: BOOL;
	xBascEntradaRecuada: BOOL;
	xBascEntradaAvancada: BOOL;
	xBascEntradaRecuando: BOOL;
	xBascEntradaAvancando: BOOL;
	xMeBascEntrAvanco: BOOL;
	xMeBascEntrRecuo: BOOL;
END_VAR

(*---------------- ENTRADAS ---------------*)
(* xBtAvancMesaBascul = Botão Levanta Mesa*)
(* xBtRecuoMesaBascul = Botão Abaixa Mesa*)
(* xS01PistPneumRecuado = Sensor Pistão Pneumático Recuado*)
(* xS02PistPneumAvancad = Sensor Pistão Pneumático Atuado*)
(* xS03PistHidraulRecuado = Sensor Pistão Hidraulico Recuado*)
(* xS04PistHidraulAvancad = Sensor Pistão Hidraulico Avanção*)
(* xS05NivelaSubida = Sensor Pistão Hidraulico Nivela Inferior*)
(* xS06NivelaDescida = Sensor Pistão Hidraulico Nivela Superior*)

(*----------------- SAÍDAS -----------------*)
(* xValvulaAbreBraco=  Válvula Acionamento do Pistão Pneumático Abertura do Braço*)
(* xValvulaFechBraco=  Válvula Acionamento do Pistão Pneumático Fechamento do Braço*)
(* xValvulaAvancPneum = Válvula Acionamento do Pistão Pneumático Sobe Mesa*)
(* xValvulaRecuaPneum = Válvula Acionamento do Pistão Pneumático Sobe Mesa*)
(* xValvulaAvancHidra = Válvula Acionamento do Pistão Avanço Hidraulico*)
(* xValvulaRecuoHidra = Válvula Acionamento do Pistão Recuo Hidraulico*)
(* xMotorBombaHidraulica = Acionamento Bomba Hidraulica*)

IF xValvulaGradeEntrada THEN

CASE PassoMesaBasculEnt OF

	0: IF xBtAvancMesaBascul THEN
			PassoMesaBasculEnt:=1;
		END_IF
		IF xBtRecuoMesaBascul THEN
			PassoMesaBasculEnt:=3;
		END_IF

	1:	IF xS01PistPneumRecuado AND xS03PistHidraulRecuado THEN
			PassoMesaBasculEnt:=5;
		ELSE
			PassoMesaBasculEnt:=0;
		END_IF

	3:	IF NOT xS01PistPneumRecuado AND NOT xS03PistHidraulRecuado THEN
			PassoMesaBasculEnt:=4;
		ELSE
			PassoMesaBasculEnt:=0;
		END_IF

	4:	xValvulaRecuoHidra:=TRUE;
		IF xS06NivelaDescida THEN
			PassoMesaBasculEnt:=60;
		END_IF
		IF xS05NivelaSubida THEN
			PassoMesaBasculEnt:=0;
		END_IF

	5:	xValvulaAbreBraco:=TRUE;
		TonAbreBracoIn:=TRUE;
		xMeBascEntrAvanco:=TRUE;
		PassoMesaBasculEnt:=10;

	10:	IF 	TonAbreBracoQ THEN
			PassoMesaBasculEnt:=15;
		END_IF
		IF	xBtRecuoMesaBascul THEN
			PassoMesaBasculEnt:=11;
		END_IF

	11: xValvulaAbreBraco:=FALSE;
		TonAbreBracoIn:=FALSE;
		PassoMesaBasculEnt:=12;

	12:	xMeBascEntrAvanco:=FALSE;
		xMeBascEntrRecuo:=TRUE;
		xValvulaFechBraco:=TRUE;
		TonFechaBracoIn:=TRUE;
		PassoMesaBasculEnt:=13;

	13:IF TonFechaBracoQ OR xBtAvancMesaBascul THEN
			PassoMesaBasculEnt:=14;
		END_IF

	14:	xValvulaFechBraco:=FALSE;
		TonFechaBracoIn:=FALSE;
		xMeBascEntrAvanco:=FALSE;
		xMeBascEntrRecuo:=FALSE;
		PassoMesaBasculEnt:=0;

	15:	xValvulaAbreBraco:=FALSE;
		TonAbreBracoIn:=FALSE;
		PassoMesaBasculEnt:=20;

	20:	xValvulaAvancHidra:=xBtAvancMesaBascul;
		IF	xS05NivelaSubida THEN
			PassoMesaBasculEnt:=25;
		END_IF
		IF	xBtRecuoMesaBascul THEN
			PassoMesaBasculEnt:=12;
		END_IF

	25:	xValvulaAvancHidra:=xBtAvancMesaBascul;
		xValvulaAvancPneum:=TRUE;
		PassoMesaBasculEnt:=30;

	30:	xValvulaAvancHidra:=xBtAvancMesaBascul;
		IF	xS02PistPneumAvancad THEN
			PassoMesaBasculEnt:=35;
		END_IF

	35:	xValvulaAvancPneum:=FALSE;
		PassoMesaBasculEnt:=40;

	40:	xValvulaAvancHidra:=xBtAvancMesaBascul;
		IF	xS04PistHidraulAvancad THEN
			PassoMesaBasculEnt:=45;
		END_IF
		IF xBtRecuoMesaBascul THEN
			PassoMesaBasculEnt:=50;
		END_IF

	45:	xValvulaAvancHidra:=FALSE;
		xMeBascEntrAvanco:=FALSE;
		PassoMesaBasculEnt:=50;

	50:	IF xBtRecuoMesaBascul THEN
			PassoMesaBasculEnt:=52;
		END_IF

	52:	xMeBascEntrAvanco:=FALSE;
		xMeBascEntrRecuo:=TRUE;
		PassoMesaBasculEnt:=55;

	55:	xValvulaRecuoHidra:=xBtRecuoMesaBascul;
		IF	xS06NivelaDescida THEN
			PassoMesaBasculEnt:=60;
		END_IF
		IF xBtAvancMesaBascul THEN
			PassoMesaBasculEnt:=56;
		END_IF

	56:	xMeBascEntrAvanco:=TRUE;
		xMeBascEntrRecuo:=FALSE;
		PassoMesaBasculEnt:=40;

	60:	xValvulaRecuoHidra:=TRUE;
		xValvulaFechBraco:=TRUE;
		TonFechaBracoIn:=TRUE;
		PassoMesaBasculEnt:=65;

	65:	IF	xS03PistHidraulRecuado THEN
			xValvulaRecuoHidra:=FALSE;
		END_IF
		IF	TonFechaBracoQ THEN
			PassoMesaBasculEnt:=70;
		END_IF

	70:	xValvulaFechBraco:=FALSE;
		TonFechaBracoIn:=FALSE;
		PassoMesaBasculEnt:=75;

	75:	xValvulaRecuaPneum:=TRUE;
		PassoMesaBasculEnt:=80;

	80:	IF xS01PistPneumRecuado THEN
			xValvulaRecuaPneum:=FALSE;
		END_IF
		IF	xS03PistHidraulRecuado THEN
			xValvulaRecuoHidra:=FALSE;
		END_IF
		IF 	xS01PistPneumRecuado AND xS03PistHidraulRecuado THEN
			PassoMesaBasculEnt:=81;
		END_IF

	81:	xMeBascEntrRecuo:=FALSE;
		PassoMesaBasculEnt:=0;

END_CASE
END_IF

TonAbreBraco(IN:= TonAbreBracoIn, PT:=T#10S , Q=> TonAbreBracoQ, ET=> );
TonFechaBraco(IN:= TonFechaBracoIn, PT:=T#10S , Q=> TonFechaBracoQ, ET=> );

IF xS01PistPneumRecuado AND xS03PistHidraulRecuado THEN
	xBascEntradaRecuada:=TRUE;
ELSE
	xBascEntradaRecuada:=FALSE;
END_IF

IF xS02PistPneumAvancad AND xS04PistHidraulAvancad THEN
	xBascEntradaAvancada:=TRUE;
ELSE
	xBascEntradaAvancada:=FALSE;
END_IF

xBascEntradaAvancando:=xMeBascEntrAvanco;
xBascEntradaRecuando:=xMeBascEntrRecuo;

IF xBascEntradaRecuada THEN
	iStatusBasculanteEntrada:=1;
END_IF
IF xBascEntradaAvancando THEN
	iStatusBasculanteEntrada:=2;
END_IF
IF xBascEntradaAvancada THEN
	iStatusBasculanteEntrada:=3;
END_IF
IF xBascEntradaRecuando THEN
	iStatusBasculanteEntrada:=4;
END_IF

(* ---- O_Portas.prg.st ---- *)
PROGRAM O_Portas
VAR
	PortaEntradaForno: HabilitaDesabilita;
	PortaSaidaForno: HabilitaDesabilita;
END_VAR

PortaEntradaForno(
	Entrada:= xBtAbrePortaEntradaForno,
	Entrada02:= ,
	Entrada03:= xOperacaoManual,
	Alarme01:= ,
	Alarme02:= ,
	Alarme03:= ,
	StatusSaida=> xPortaEntradaFornoForce);

IF xBtAbrePortaEntradaForno THEN
	xBtAbrePortaEntradaForno:=FALSE;
END_IF

PortaSaidaForno(
	Entrada:= xBtAbrePortaSaidaForno,
	Entrada02:= ,
	Entrada03:= xOperacaoManual,
	Alarme01:= ,
	Alarme02:= ,
	Alarme03:= ,
	StatusSaida=> xPortaSaidaFornoForce);

IF xBtAbrePortaSaidaForno THEN
	xBtAbrePortaSaidaForno:=FALSE;
END_IF

xValvPortaEntradaForno:= NOT (xPortaEntradaForno	OR xPortaEntradaFornoForce OR xOperacaoManual);
xValvPortaSaidaForno:=	NOT (xPortaSaidaForno OR xPortaSaidaFornoForce OR xOperacaoManual);
